LIN {X 0,Y 319.626,Z 323.132,A -85,B 0,C 180,E1 -15102.071,E2 -15102.071} C_VEL
LIN {X 0,Y 319.734,Z 323.151,A -85,B 0,C 180,E1 -15106.008,E2 -15106.008} C_VEL
LIN {X 0,Y 319.737,Z 323.147,A -85,B 0,C 180,E1 -15109.872,E2 -15109.872} C_VEL
LIN {X 0,Y 319.902,Z 323.101,A -85,B 0,C 180,E1 -15113.693,E2 -15113.693} C_VEL
LIN {X 0,Y 319.959,Z 323.12,A -85,B 0,C 180,E1 -15117.482,E2 -15117.482} C_VEL
LIN {X 0,Y 320.015,Z 323.113,A -85,B 0,C 180,E1 -15121.258,E2 -15121.258} C_VEL
LIN {X 0,Y 319.917,Z 323.111,A -85,B 0,C 180,E1 -15126.306,E2 -15126.306} C_VEL
LIN {X 0,Y 319.737,Z 323.154,A -85,B 0,C 180,E1 -15130.127,E2 -15130.127} C_VEL
LIN {X 0,Y 319.71,Z 323.137,A -85,B 0,C 180,E1 -15133.993,E2 -15133.993} C_VEL
LIN {X 0,Y 319.587,Z 323.169,A -85,B 0,C 180,E1 -15137.931,E2 -15137.931} C_VEL
LIN {X 0,Y 319.564,Z 323.172,A -85,B 0,C 180,E1 -15141.954,E2 -15141.954} C_VEL
LIN {X 0,Y 319.567,Z 323.17,A -85,B 0,C 180,E1 -15146.094,E2 -15146.094} C_VEL
LIN {X 0,Y 319.541,Z 323.179,A -85,B 0,C 180,E1 -15148.938,E2 -15148.938} C_VEL
LIN {X 0,Y 319.523,Z 323.172,A -85,B 0,C 180,E1 -15151.862,E2 -15151.862} C_VEL
LIN {X 0,Y 319.579,Z 323.174,A -85,B 0,C 180,E1 -15155.542,E2 -15155.542} C_VEL
LIN {X 0,Y 319.527,Z 323.183,A -85,B 0,C 180,E1 -15159.661,E2 -15159.661} C_VEL
LIN {X 0,Y 319.517,Z 323.178,A -85,B 0,C 180,E1 -15163.459,E2 -15163.459} C_VEL
LIN {X 0,Y 319.548,Z 323.18,A -85,B 0,C 180,E1 -15167.015,E2 -15167.015} C_VEL
LIN {X 0,Y 319.543,Z 323.181,A -85,B 0,C 180,E1 -15170.37,E2 -15170.37} C_VEL
LIN {X 0,Y 319.577,Z 323.176,A -85,B 0,C 180,E1 -15174.457,E2 -15174.457} C_VEL
LIN {X 0,Y 319.522,Z 323.186,A -85,B 0,C 180,E1 -15178.137,E2 -15178.137} C_VEL
LIN {X 0,Y 319.566,Z 323.328,A -85,B 0,C 180,E1 -15179.059,E2 -15179.059} C_VEL
LIN {X 0,Y 321.759,Z 333.663,A -85,B 0,C 180,E1 -15182.344,E2 -15182.344} C_VEL
LIN {X 0,Y 323.542,Z 343.466,A -85,B 0,C 180,E1 -15185.283,E2 -15185.283} C_VEL
LIN {X 0,Y 323.619,Z 344.48,A -85,B 0,C 180,E1 -15185.48,E2 -15185.48} C_VEL
LIN {X 0,Y 328.326,Z 371.476,A -85,B 0,C 180,E1 -15186.494,E2 -15186.494} C_VEL
LIN {X 0,Y 329.76,Z 380.86,A -85,B 0,C 180,E1 -15186.815,E2 -15186.815} C_VEL
LIN {X 0,Y 328.137,Z 450.866,A -85,B 0,C 180,E1 -15188.401,E2 -15188.401} C_VEL
LIN {X 0,Y 327.713,Z 460.449,A -85,B 0,C 180,E1 -15188.742,E2 -15188.742} C_VEL
LIN {X 0,Y 327.027,Z 470.32,A -85,B 0,C 180,E1 -15189.231,E2 -15189.231} C_VEL
LIN {X 0,Y 326.274,Z 479.678,A -85,B 0,C 180,E1 -15189.84,E2 -15189.84} C_VEL
LIN {X 0,Y 325.191,Z 490.522,A -85,B 0,C 180,E1 -15190.756,E2 -15190.756} C_VEL
LIN {X 0,Y 324.039,Z 500.641,A -85,B 0,C 180,E1 -15191.834,E2 -15191.834} C_VEL
LIN {X 0,Y 322.955,Z 509.479,A -85,B 0,C 180,E1 -15192.981,E2 -15192.981} C_VEL
LIN {X 0,Y 321.975,Z 517.57,A -85,B 0,C 180,E1 -15194.242,E2 -15194.242} C_VEL
LIN {X 0,Y 320.934,Z 525.527,A -85,B 0,C 180,E1 -15195.738,E2 -15195.738} C_VEL
LIN {X 0,Y 319.888,Z 532.482,A -85,B 0,C 180,E1 -15197.308,E2 -15197.308} C_VEL
LIN {X 0,Y 319.042,Z 539.265,A -85,B 0,C 180,E1 -15199.208,E2 -15199.208} C_VEL
LIN {X 0,Y 318.623,Z 543.11,A -85,B 0,C 180,E1 -15200.478,E2 -15200.478} C_VEL
LIN {X 0,Y 318.164,Z 547.736,A -85,B 0,C 180,E1 -15202.384,E2 -15202.384} C_VEL
LIN {X 0,Y 317.864,Z 551.156,A -85,B 0,C 180,E1 -15204.237,E2 -15204.237} C_VEL
LIN {X 0,Y 317.772,Z 553.736,A -85,B 0,C 180,E1 -15206.196,E2 -15206.196} C_VEL
LIN {X 0,Y 317.686,Z 555.558,A -85,B 0,C 180,E1 -15208.732,E2 -15208.732} C_VEL
LIN {X 0,Y 317.7,Z 555.874,A -85,B 0,C 180,E1 -15210,E2 -15210} C_VEL
LIN {X 0,Y 317.725,Z 555.365,A -85,B 0,C 180,E1 -15212.535,E2 -15212.535} C_VEL
LIN {X 0,Y 317.843,Z 553.108,A -85,B 0,C 180,E1 -15215.074,E2 -15215.074} C_VEL
LIN {X 0,Y 318.061,Z 550.377,A -85,B 0,C 180,E1 -15216.98,E2 -15216.98} C_VEL
LIN {X 0,Y 318.49,Z 546.623,A -85,B 0,C 180,E1 -15218.886,E2 -15218.886} C_VEL
LIN {X 0,Y 319.153,Z 541.741,A -85,B 0,C 180,E1 -15220.788,E2 -15220.788} C_VEL
LIN {X 0,Y 319.861,Z 536.759,A -85,B 0,C 180,E1 -15222.37,E2 -15222.37} C_VEL
LIN {X 0,Y 321.147,Z 529.338,A -85,B 0,C 180,E1 -15224.252,E2 -15224.252} C_VEL
LIN {X 0,Y 322.305,Z 521.825,A -85,B 0,C 180,E1 -15225.817,E2 -15225.817} C_VEL
LIN {X 0,Y 323.459,Z 513.882,A -85,B 0,C 180,E1 -15227.195,E2 -15227.195} C_VEL
LIN {X 0,Y 324.723,Z 505.12,A -85,B 0,C 180,E1 -15228.453,E2 -15228.453} C_VEL
LIN {X 0,Y 325.995,Z 496.099,A -85,B 0,C 180,E1 -15229.521,E2 -15229.521} C_VEL
LIN {X 0,Y 327.231,Z 486.747,A -85,B 0,C 180,E1 -15230.426,E2 -15230.426} C_VEL
LIN {X 0,Y 328.338,Z 475.986,A -85,B 0,C 180,E1 -15231.256,E2 -15231.256} C_VEL
LIN {X 0,Y 329.341,Z 464.293,A -85,B 0,C 180,E1 -15231.928,E2 -15231.928} C_VEL
LIN {X 0,Y 330.1,Z 453.228,A -85,B 0,C 180,E1 -15232.369,E2 -15232.369} C_VEL
LIN {X 0,Y 330.612,Z 433.555,A -85,B 0,C 180,E1 -15232.868,E2 -15232.868} C_VEL
LIN {X 0,Y 331.874,Z 381.21,A -85,B 0,C 180,E1 -15234.044,E2 -15234.044} C_VEL
LIN {X 0,Y 328.247,Z 359.793,A -85,B 0,C 180,E1 -15234.893,E2 -15234.893} C_VEL
LIN {X 0,Y 325.512,Z 347.56,A -85,B 0,C 180,E1 -15235.451,E2 -15235.451} C_VEL
LIN {X 0,Y 323.992,Z 343.545,A -85,B 0,C 180,E1 -15235.749,E2 -15235.749} C_VEL
LIN {X 0,Y 321.996,Z 333.704,A -85,B 0,C 180,E1 -15238.697,E2 -15238.697} C_VEL
LIN {X 0,Y 319.726,Z 323.984,A -85,B 0,C 180,E1 -15241.84,E2 -15241.84} C_VEL
LIN {X 0,Y 319.563,Z 323.201,A -85,B 0,C 180,E1 -15242.23,E2 -15242.23} C_VEL
LIN {X 0,Y 319.557,Z 323.173,A -85,B 0,C 180,E1 -15246.428,E2 -15246.428} C_VEL
LIN {X 0,Y 319.557,Z 323.169,A -85,B 0,C 180,E1 -15249.669,E2 -15249.669} C_VEL
LIN {X 0,Y 319.519,Z 323.183,A -85,B 0,C 180,E1 -15253.461,E2 -15253.461} C_VEL
LIN {X 0,Y 319.552,Z 323.18,A -85,B 0,C 180,E1 -15257.017,E2 -15257.017} C_VEL
LIN {X 0,Y 319.545,Z 323.179,A -85,B 0,C 180,E1 -15260.371,E2 -15260.371} C_VEL
LIN {X 0,Y 319.578,Z 323.17,A -85,B 0,C 180,E1 -15264.457,E2 -15264.457} C_VEL
LIN {X 0,Y 319.53,Z 323.177,A -85,B 0,C 180,E1 -15268.139,E2 -15268.139} C_VEL
LIN {X 0,Y 319.61,Z 323.169,A -85,B 0,C 180,E1 -15271.591,E2 -15271.591} C_VEL
LIN {X 0,Y 319.605,Z 323.171,A -85,B 0,C 180,E1 -15275.304,E2 -15275.304} C_VEL
LIN {X 0,Y 319.597,Z 323.169,A -85,B 0,C 180,E1 -15278.048,E2 -15278.048} C_VEL
LIN {X 0,Y 319.689,Z 323.156,A -85,B 0,C 180,E1 -15280.962,E2 -15280.962} C_VEL
LIN {X 0,Y 319.731,Z 323.152,A -85,B 0,C 180,E1 -15285.276,E2 -15285.276} C_VEL
LIN {X 0,Y 319.759,Z 323.149,A -85,B 0,C 180,E1 -15289.873,E2 -15289.873} C_VEL
LIN {X 0,Y 319.935,Z 323.13,A -85,B 0,C 180,E1 -15292.427,E2 -15292.427} C_VEL
LIN {X 0,Y 319.749,Z 323.148,A -85,B 0,C 180,E1 -15294.956,E2 -15294.956} C_VEL
LIN {X 0,Y 319.993,Z 323.122,A -85,B 0,C 180,E1 -15297.483,E2 -15297.483} C_VEL
LIN {X 0,Y 320.152,Z 323.098,A -85,B 0,C 180,E1 -15300,E2 -15300} C_VEL
LIN {X 0,Y 319.993,Z 323.125,A -85,B 0,C 180,E1 -15302.518,E2 -15302.518} C_VEL
LIN {X 0,Y 319.934,Z 323.128,A -85,B 0,C 180,E1 -15306.628,E2 -15306.628} C_VEL
LIN {X 0,Y 319.759,Z 323.152,A -85,B 0,C 180,E1 -15310.127,E2 -15310.127} C_VEL
LIN {X 0,Y 319.732,Z 323.156,A -85,B 0,C 180,E1 -15314.724,E2 -15314.724} C_VEL
LIN {X 0,Y 319.69,Z 323.158,A -85,B 0,C 180,E1 -15319.038,E2 -15319.038} C_VEL
LIN {X 0,Y 319.559,Z 323.179,A -85,B 0,C 180,E1 -15323.321,E2 -15323.321} C_VEL
LIN {X 0,Y 319.589,Z 323.175,A -85,B 0,C 180,E1 -15326.092,E2 -15326.092} C_VEL
LIN {X 0,Y 319.576,Z 323.173,A -85,B 0,C 180,E1 -15328.935,E2 -15328.935} C_VEL
LIN {X 0,Y 319.531,Z 323.177,A -85,B 0,C 180,E1 -15331.862,E2 -15331.862} C_VEL
LIN {X 0,Y 319.57,Z 323.179,A -85,B 0,C 180,E1 -15335.54,E2 -15335.54} C_VEL
LIN {X 0,Y 319.649,Z 323.459,A -85,B 0,C 180,E1 -15336.347,E2 -15336.347} C_VEL
LIN {X 0,Y 322.123,Z 333.874,A -85,B 0,C 180,E1 -15339.665,E2 -15339.665} C_VEL
LIN {X 0,Y 322.612,Z 336.041,A -85,B 0,C 180,E1 -15340.207,E2 -15340.207} C_VEL
LIN {X 0,Y 328.68,Z 350.643,A -85,B 0,C 180,E1 -15341.162,E2 -15341.162} C_VEL
LIN {X 0,Y 332.144,Z 368.395,A -85,B 0,C 180,E1 -15341.908,E2 -15341.908} C_VEL
LIN {X 0,Y 330.201,Z 442.436,A -85,B 0,C 180,E1 -15343.6,E2 -15343.6} C_VEL
LIN {X 0,Y 329.689,Z 451.952,A -85,B 0,C 180,E1 -15343.936,E2 -15343.936} C_VEL
LIN {X 0,Y 329.089,Z 461.748,A -85,B 0,C 180,E1 -15344.432,E2 -15344.432} C_VEL
LIN {X 0,Y 328.119,Z 472.227,A -85,B 0,C 180,E1 -15345.131,E2 -15345.131} C_VEL
LIN {X 0,Y 327.138,Z 481.657,A -85,B 0,C 180,E1 -15345.931,E2 -15345.931} C_VEL
LIN {X 0,Y 325.754,Z 492.603,A -85,B 0,C 180,E1 -15347.108,E2 -15347.108} C_VEL
LIN {X 0,Y 324.528,Z 501.273,A -85,B 0,C 180,E1 -15348.247,E2 -15348.247} C_VEL
LIN {X 0,Y 323.167,Z 509.632,A -85,B 0,C 180,E1 -15349.566,E2 -15349.566} C_VEL
LIN {X 0,Y 321.945,Z 517.518,A -85,B 0,C 180,E1 -15351.082,E2 -15351.082} C_VEL
LIN {X 0,Y 320.914,Z 524.004,A -85,B 0,C 180,E1 -15352.575,E2 -15352.575} C_VEL
LIN {X 0,Y 319.836,Z 530.455,A -85,B 0,C 180,E1 -15354.393,E2 -15354.393} C_VEL
LIN {X 0,Y 319.231,Z 534.761,A -85,B 0,C 180,E1 -15355.848,E2 -15355.848} C_VEL
LIN {X 0,Y 318.47,Z 539.726,A -85,B 0,C 180,E1 -15358.02,E2 -15358.02} C_VEL
LIN {X 0,Y 318.152,Z 542.372,A -85,B 0,C 180,E1 -15359.487,E2 -15359.487} C_VEL
LIN {X 0,Y 317.871,Z 544.215,A -85,B 0,C 180,E1 -15360.895,E2 -15360.895} C_VEL
LIN {X 0,Y 317.665,Z 545.633,A -85,B 0,C 180,E1 -15362.316,E2 -15362.316} C_VEL
LIN {X 0,Y 317.493,Z 546.626,A -85,B 0,C 180,E1 -15363.723,E2 -15363.723} C_VEL
LIN {X 0,Y 317.423,Z 546.993,A -85,B 0,C 180,E1 -15365.2,E2 -15365.2} C_VEL
LIN {X 0,Y 317.434,Z 546.413,A -85,B 0,C 180,E1 -15367.89,E2 -15367.89} C_VEL
LIN {X 0,Y 317.593,Z 545.359,A -85,B 0,C 180,E1 -15369.264,E2 -15369.264} C_VEL
LIN {X 0,Y 317.987,Z 541.947,A -85,B 0,C 180,E1 -15371.976,E2 -15371.976} C_VEL
LIN {X 0,Y 318.387,Z 538.074,A -85,B 0,C 180,E1 -15373.983,E2 -15373.983} C_VEL
LIN {X 0,Y 318.979,Z 532.982,A -85,B 0,C 180,E1 -15375.974,E2 -15375.974} C_VEL
LIN {X 0,Y 319.643,Z 527.744,A -85,B 0,C 180,E1 -15377.621,E2 -15377.621} C_VEL
LIN {X 0,Y 320.481,Z 521.404,A -85,B 0,C 180,E1 -15379.257,E2 -15379.257} C_VEL
LIN {X 0,Y 321.607,Z 513.482,A -85,B 0,C 180,E1 -15380.922,E2 -15380.922} C_VEL
LIN {X 0,Y 322.656,Z 505.376,A -85,B 0,C 180,E1 -15382.333,E2 -15382.333} C_VEL
LIN {X 0,Y 323.8,Z 496.471,A -85,B 0,C 180,E1 -15383.614,E2 -15383.614} C_VEL
LIN {X 0,Y 324.744,Z 488.557,A -85,B 0,C 180,E1 -15384.573,E2 -15384.573} C_VEL
LIN {X 0,Y 325.898,Z 477.255,A -85,B 0,C 180,E1 -15385.671,E2 -15385.671} C_VEL
LIN {X 0,Y 326.86,Z 466.957,A -85,B 0,C 180,E1 -15386.456,E2 -15386.456} C_VEL
LIN {X 0,Y 327.52,Z 456.409,A -85,B 0,C 180,E1 -15387.079,E2 -15387.079} C_VEL
LIN {X 0,Y 328.185,Z 445.003,A -85,B 0,C 180,E1 -15387.545,E2 -15387.545} C_VEL
LIN {X 0,Y 328.673,Z 428.296,A -85,B 0,C 180,E1 -15387.971,E2 -15387.971} C_VEL
LIN {X 0,Y 329.901,Z 367.398,A -85,B 0,C 180,E1 -15389.329,E2 -15389.329} C_VEL
LIN {X 0,Y 325.686,Z 345.307,A -85,B 0,C 180,E1 -15390.151,E2 -15390.151} C_VEL
LIN {X 0,Y 322.567,Z 336.108,A -85,B 0,C 180,E1 -15390.648,E2 -15390.648} C_VEL
LIN {X 0,Y 320.926,Z 328.238,A -85,B 0,C 180,E1 -15393.139,E2 -15393.139} C_VEL
LIN {X 0,Y 319.738,Z 323.207,A -85,B 0,C 180,E1 -15394.886,E2 -15394.886} C_VEL
LIN {X 0,Y 319.937,Z 323.128,A -85,B 0,C 180,E1 -15396.306,E2 -15396.306} C_VEL
LIN {X 0,Y 319.737,Z 323.157,A -85,B 0,C 180,E1 -15400.128,E2 -15400.128} C_VEL
LIN {X 0,Y 319.734,Z 323.158,A -85,B 0,C 180,E1 -15403.992,E2 -15403.992} C_VEL
LIN {X 0,Y 319.66,Z 323.165,A -85,B 0,C 180,E1 -15407.927,E2 -15407.927} C_VEL
LIN {X 0,Y 319.605,Z 323.176,A -85,B 0,C 180,E1 -15410.6,E2 -15410.6} C_VEL
LIN {X 0,Y 319.606,Z 323.171,A -85,B 0,C 180,E1 -15414.696,E2 -15414.696} C_VEL
LIN {X 0,Y 319.613,Z 323.16,A -85,B 0,C 180,E1 -15418.41,E2 -15418.41} C_VEL
LIN {X 0,Y 319.532,Z 323.179,A -85,B 0,C 180,E1 -15421.862,E2 -15421.862} C_VEL
LIN {X 0,Y 319.548,Z 323.162,A -85,B 0,C 180,E1 -15424.612,E2 -15424.612} C_VEL
LIN {X 0,Y 318.92,Z 323.25,A -85,B 0,C 180,E1 -15425.664,E2 -15425.664} C_VEL
LIN {X 0,Y 316.093,Z 323.61,A -85,B 0,C 180,E1 -15427.378,E2 -15427.378} C_VEL
LIN {X 0,Y 313.662,Z 323.912,A -85,B 0,C 180,E1 -15428.766,E2 -15428.766} C_VEL
LIN {X 0,Y 312.598,Z 324.039,A -85,B 0,C 180,E1 -15429.841,E2 -15429.841} C_VEL
LIN {X 0,Y 312.502,Z 324.045,A -85,B 0,C 180,E1 -15430.206,E2 -15430.206} C_VEL
LIN {X 0,Y 312.475,Z 324.055,A -85,B 0,C 180,E1 -15434.206,E2 -15434.206} C_VEL
LIN {X 0,Y 312.486,Z 324.053,A -85,B 0,C 180,E1 -15437.919,E2 -15437.919} C_VEL
LIN {X 0,Y 312.479,Z 324.035,A -85,B 0,C 180,E1 -15440.968,E2 -15440.968} C_VEL
LIN {X 0,Y 312.533,Z 324.05,A -85,B 0,C 180,E1 -15444.22,E2 -15444.22} C_VEL
LIN {X 0,Y 312.503,Z 324.052,A -85,B 0,C 180,E1 -15447.333,E2 -15447.333} C_VEL
LIN {X 0,Y 312.509,Z 324.024,A -85,B 0,C 180,E1 -15451.291,E2 -15451.291} C_VEL
LIN {X 0,Y 312.556,Z 324.049,A -85,B 0,C 180,E1 -15454.708,E2 -15454.708} C_VEL
LIN {X 0,Y 312.568,Z 324.045,A -85,B 0,C 180,E1 -15457.527,E2 -15457.527} C_VEL
LIN {X 0,Y 312.584,Z 324.008,A -85,B 0,C 180,E1 -15461.653,E2 -15461.653} C_VEL
LIN {X 0,Y 312.688,Z 324.03,A -85,B 0,C 180,E1 -15465.686,E2 -15465.686} C_VEL
LIN {X 0,Y 312.687,Z 324.028,A -85,B 0,C 180,E1 -15469.641,E2 -15469.641} C_VEL
LIN {X 0,Y 312.798,Z 323.991,A -85,B 0,C 180,E1 -15472.252,E2 -15472.252} C_VEL
LIN {X 0,Y 312.692,Z 324.007,A -85,B 0,C 180,E1 -15474.842,E2 -15474.842} C_VEL
LIN {X 0,Y 312.969,Z 323.998,A -85,B 0,C 180,E1 -15478.713,E2 -15478.713} C_VEL
LIN {X 0,Y 312.982,Z 323.989,A -85,B 0,C 180,E1 -15481.286,E2 -15481.286} C_VEL
LIN {X 0,Y 312.86,Z 323.99,A -85,B 0,C 180,E1 -15486.449,E2 -15486.449} C_VEL
LIN {X 0,Y 312.752,Z 324.024,A -85,B 0,C 180,E1 -15489.05,E2 -15489.05} C_VEL
LIN {X 0,Y 312.626,Z 324.033,A -85,B 0,C 180,E1 -15492.991,E2 -15492.991} C_VEL
LIN {X 0,Y 312.57,Z 324.024,A -85,B 0,C 180,E1 -15495.653,E2 -15495.653} C_VEL
LIN {X 0,Y 312.534,Z 324.054,A -85,B 0,C 180,E1 -15499.712,E2 -15499.712} C_VEL
LIN {X 0,Y 312.521,Z 324.038,A -85,B 0,C 180,E1 -15502.777,E2 -15502.777} C_VEL
LIN {X 0,Y 312.528,Z 324.046,A -85,B 0,C 180,E1 -15505.907,E2 -15505.907} C_VEL
LIN {X 0,Y 312.495,Z 324.05,A -85,B 0,C 180,E1 -15509.655,E2 -15509.655} C_VEL
LIN {X 0,Y 312.519,Z 324.058,A -85,B 0,C 180,E1 -15513.688,E2 -15513.688} C_VEL
LIN {X 0,Y 312.51,Z 324.046,A -85,B 0,C 180,E1 -15517.387,E2 -15517.387} C_VEL
LIN {X 0,Y 312.439,Z 324.063,A -85,B 0,C 180,E1 -15520.717,E2 -15520.717} C_VEL
LIN {X 0,Y 312.448,Z 324.065,A -85,B 0,C 180,E1 -15524.21,E2 -15524.21} C_VEL
LIN {X 0,Y 312.452,Z 324.064,A -85,B 0,C 180,E1 -15527.925,E2 -15527.925} C_VEL
LIN {X 0,Y 312.482,Z 324.058,A -85,B 0,C 180,E1 -15531.922,E2 -15531.922} C_VEL
LIN {X 0,Y 312.528,Z 324.054,A -85,B 0,C 180,E1 -15534.22,E2 -15534.22} C_VEL
LIN {X 0,Y 312.476,Z 324.064,A -85,B 0,C 180,E1 -15538.088,E2 -15538.088} C_VEL
LIN {X 0,Y 312.525,Z 324.325,A -85,B 0,C 180,E1 -15538.708,E2 -15538.708} C_VEL
LIN {X 0,Y 314.721,Z 334.563,A -85,B 0,C 180,E1 -15542.034,E2 -15542.034} C_VEL
LIN {X 0,Y 316.54,Z 344.066,A -85,B 0,C 180,E1 -15544.917,E2 -15544.917} C_VEL
LIN {X 0,Y 317.353,Z 347.388,A -85,B 0,C 180,E1 -15545.128,E2 -15545.128} C_VEL
LIN {X 0,Y 322.634,Z 377.952,A -85,B 0,C 180,E1 -15546.256,E2 -15546.256} C_VEL
LIN {X 0,Y 323.125,Z 381.869,A -85,B 0,C 180,E1 -15546.386,E2 -15546.386} C_VEL
LIN {X 0,Y 321.461,Z 450.859,A -85,B 0,C 180,E1 -15547.982,E2 -15547.982} C_VEL
LIN {X 0,Y 321.033,Z 460.207,A -85,B 0,C 180,E1 -15548.32,E2 -15548.32} C_VEL
LIN {X 0,Y 320.267,Z 470.718,A -85,B 0,C 180,E1 -15548.856,E2 -15548.856} C_VEL
LIN {X 0,Y 319.396,Z 480.902,A -85,B 0,C 180,E1 -15549.554,E2 -15549.554} C_VEL
LIN {X 0,Y 318.295,Z 491.487,A -85,B 0,C 180,E1 -15550.49,E2 -15550.49} C_VEL
LIN {X 0,Y 317.092,Z 501.414,A -85,B 0,C 180,E1 -15551.589,E2 -15551.589} C_VEL
LIN {X 0,Y 316.054,Z 509.696,A -85,B 0,C 180,E1 -15552.697,E2 -15552.697} C_VEL
LIN {X 0,Y 315.051,Z 517.587,A -85,B 0,C 180,E1 -15553.958,E2 -15553.958} C_VEL
LIN {X 0,Y 314.017,Z 525.219,A -85,B 0,C 180,E1 -15555.417,E2 -15555.417} C_VEL
LIN {X 0,Y 312.953,Z 532.212,A -85,B 0,C 180,E1 -15557.022,E2 -15557.022} C_VEL
LIN {X 0,Y 312.047,Z 539.027,A -85,B 0,C 180,E1 -15558.963,E2 -15558.963} C_VEL
LIN {X 0,Y 311.408,Z 544.485,A -85,B 0,C 180,E1 -15560.91,E2 -15560.91} C_VEL
LIN {X 0,Y 310.95,Z 548.753,A -85,B 0,C 180,E1 -15562.859,E2 -15562.859} C_VEL
LIN {X 0,Y 310.719,Z 551.951,A -85,B 0,C 180,E1 -15564.809,E2 -15564.809} C_VEL
LIN {X 0,Y 310.687,Z 553.581,A -85,B 0,C 180,E1 -15566.109,E2 -15566.109} C_VEL
LIN {X 0,Y 310.603,Z 555.448,A -85,B 0,C 180,E1 -15568.703,E2 -15568.703} C_VEL
LIN {X 0,Y 310.614,Z 555.764,A -85,B 0,C 180,E1 -15570,E2 -15570} C_VEL
LIN {X 0,Y 310.651,Z 555.291,A -85,B 0,C 180,E1 -15572.593,E2 -15572.593} C_VEL
LIN {X 0,Y 310.763,Z 553.062,A -85,B 0,C 180,E1 -15575.19,E2 -15575.19} C_VEL
LIN {X 0,Y 311.003,Z 550.354,A -85,B 0,C 180,E1 -15577.14,E2 -15577.14} C_VEL
LIN {X 0,Y 311.449,Z 546.623,A -85,B 0,C 180,E1 -15579.088,E2 -15579.088} C_VEL
LIN {X 0,Y 312.165,Z 541.766,A -85,B 0,C 180,E1 -15581.032,E2 -15581.032} C_VEL
LIN {X 0,Y 312.908,Z 536.811,A -85,B 0,C 180,E1 -15582.649,E2 -15582.649} C_VEL
LIN {X 0,Y 314.25,Z 529.419,A -85,B 0,C 180,E1 -15584.572,E2 -15584.572} C_VEL
LIN {X 0,Y 315.459,Z 521.95,A -85,B 0,C 180,E1 -15586.17,E2 -15586.17} C_VEL
LIN {X 0,Y 316.716,Z 513.909,A -85,B 0,C 180,E1 -15587.598,E2 -15587.598} C_VEL
LIN {X 0,Y 318.014,Z 505.371,A -85,B 0,C 180,E1 -15588.857,E2 -15588.857} C_VEL
LIN {X 0,Y 319.334,Z 496.44,A -85,B 0,C 180,E1 -15589.946,E2 -15589.946} C_VEL
LIN {X 0,Y 320.623,Z 487.211,A -85,B 0,C 180,E1 -15590.867,E2 -15590.867} C_VEL
LIN {X 0,Y 321.857,Z 475.424,A -85,B 0,C 180,E1 -15591.79,E2 -15591.79} C_VEL
LIN {X 0,Y 322.852,Z 464.382,A -85,B 0,C 180,E1 -15592.435,E2 -15592.435} C_VEL
LIN {X 0,Y 323.661,Z 453.42,A -85,B 0,C 180,E1 -15592.881,E2 -15592.881} C_VEL
LIN {X 0,Y 324.195,Z 434.067,A -85,B 0,C 180,E1 -15593.385,E2 -15593.385} C_VEL
LIN {X 0,Y 325.509,Z 382.081,A -85,B 0,C 180,E1 -15594.575,E2 -15594.575} C_VEL
LIN {X 0,Y 321.867,Z 360.709,A -85,B 0,C 180,E1 -15595.451,E2 -15595.451} C_VEL
LIN {X 0,Y 319.441,Z 350.024,A -85,B 0,C 180,E1 -15595.96,E2 -15595.96} C_VEL
LIN {X 0,Y 316.817,Z 343.596,A -85,B 0,C 180,E1 -15596.426,E2 -15596.426} C_VEL
LIN {X 0,Y 315.612,Z 337.505,A -85,B 0,C 180,E1 -15598.242,E2 -15598.242} C_VEL
LIN {X 0,Y 313.325,Z 327.475,A -85,B 0,C 180,E1 -15601.532,E2 -15601.532} C_VEL
LIN {X 0,Y 312.542,Z 324.09,A -85,B 0,C 180,E1 -15602.79,E2 -15602.79} C_VEL
LIN {X 0,Y 312.534,Z 324.051,A -85,B 0,C 180,E1 -15605.95,E2 -15605.95} C_VEL
LIN {X 0,Y 312.502,Z 324.046,A -85,B 0,C 180,E1 -15610.126,E2 -15610.126} C_VEL
LIN {X 0,Y 312.456,Z 324.064,A -85,B 0,C 180,E1 -15613.965,E2 -15613.965} C_VEL
LIN {X 0,Y 312.482,Z 324.056,A -85,B 0,C 180,E1 -15617.919,E2 -15617.919} C_VEL
LIN {X 0,Y 312.497,Z 324.056,A -85,B 0,C 180,E1 -15620.971,E2 -15620.971} C_VEL
LIN {X 0,Y 312.531,Z 324.049,A -85,B 0,C 180,E1 -15624.221,E2 -15624.221} C_VEL
LIN {X 0,Y 312.503,Z 324.057,A -85,B 0,C 180,E1 -15627.334,E2 -15627.334} C_VEL
LIN {X 0,Y 312.543,Z 324.05,A -85,B 0,C 180,E1 -15631.279,E2 -15631.279} C_VEL
LIN {X 0,Y 312.585,Z 324.05,A -85,B 0,C 180,E1 -15634.711,E2 -15634.711} C_VEL
LIN {X 0,Y 312.587,Z 324.041,A -85,B 0,C 180,E1 -15637.529,E2 -15637.529} C_VEL
LIN {X 0,Y 312.639,Z 324.031,A -85,B 0,C 180,E1 -15641.657,E2 -15641.657} C_VEL
LIN {X 0,Y 312.694,Z 324.024,A -85,B 0,C 180,E1 -15645.687,E2 -15645.687} C_VEL
LIN {X 0,Y 312.703,Z 324.03,A -85,B 0,C 180,E1 -15649.642,E2 -15649.642} C_VEL
LIN {X 0,Y 312.875,Z 324.007,A -85,B 0,C 180,E1 -15652.255,E2 -15652.255} C_VEL
LIN {X 0,Y 312.719,Z 324.024,A -85,B 0,C 180,E1 -15654.843,E2 -15654.843} C_VEL
LIN {X 0,Y 312.992,Z 323.995,A -85,B 0,C 180,E1 -15658.714,E2 -15658.714} C_VEL
LIN {X 0,Y 312.992,Z 323.992,A -85,B 0,C 180,E1 -15661.287,E2 -15661.287} C_VEL
LIN {X 0,Y 312.719,Z 324.024,A -85,B 0,C 180,E1 -15665.158,E2 -15665.158} C_VEL
LIN {X 0,Y 312.874,Z 324.008,A -85,B 0,C 180,E1 -15667.746,E2 -15667.746} C_VEL
LIN {X 0,Y 312.671,Z 324.033,A -85,B 0,C 180,E1 -15671.672,E2 -15671.672} C_VEL
LIN {X 0,Y 312.701,Z 324.033,A -85,B 0,C 180,E1 -15674.888,E2 -15674.888} C_VEL
LIN {X 0,Y 312.61,Z 324.039,A -85,B 0,C 180,E1 -15679.225,E2 -15679.225} C_VEL
LIN {X 0,Y 312.526,Z 324.056,A -85,B 0,C 180,E1 -15682.78,E2 -15682.78} C_VEL
LIN {X 0,Y 312.569,Z 324.052,A -85,B 0,C 180,E1 -15685.923,E2 -15685.923} C_VEL
LIN {X 0,Y 312.537,Z 324.055,A -85,B 0,C 180,E1 -15689.651,E2 -15689.651} C_VEL
LIN {X 0,Y 312.52,Z 324.051,A -85,B 0,C 180,E1 -15693.689,E2 -15693.689} C_VEL
LIN {X 0,Y 312.565,Z 324.201,A -85,B 0,C 180,E1 -15695.676,E2 -15695.676} C_VEL
LIN {X 0,Y 315.023,Z 334.395,A -85,B 0,C 180,E1 -15699.068,E2 -15699.068} C_VEL
LIN {X 0,Y 315.399,Z 335.975,A -85,B 0,C 180,E1 -15699.477,E2 -15699.477} C_VEL
LIN {X 0,Y 322.335,Z 352.441,A -85,B 0,C 180,E1 -15700.625,E2 -15700.625} C_VEL
LIN {X 0,Y 325.131,Z 365.615,A -85,B 0,C 180,E1 -15701.22,E2 -15701.22} C_VEL
LIN {X 0,Y 325.83,Z 369.74,A -85,B 0,C 180,E1 -15701.387,E2 -15701.387} C_VEL
LIN {X 0,Y 323.775,Z 442.238,A -85,B 0,C 180,E1 -15703.067,E2 -15703.067} C_VEL
LIN {X 0,Y 323.231,Z 452.055,A -85,B 0,C 180,E1 -15703.419,E2 -15703.419} C_VEL
LIN {X 0,Y 322.593,Z 461.823,A -85,B 0,C 180,E1 -15703.921,E2 -15703.921} C_VEL
LIN {X 0,Y 321.701,Z 471.566,A -85,B 0,C 180,E1 -15704.573,E2 -15704.573} C_VEL
LIN {X 0,Y 320.586,Z 481.765,A -85,B 0,C 180,E1 -15705.451,E2 -15705.451} C_VEL
LIN {X 0,Y 319.172,Z 492.366,A -85,B 0,C 180,E1 -15706.606,E2 -15706.606} C_VEL
LIN {X 0,Y 317.843,Z 501.346,A -85,B 0,C 180,E1 -15707.807,E2 -15707.807} C_VEL
LIN {X 0,Y 316.311,Z 510.289,A -85,B 0,C 180,E1 -15709.261,E2 -15709.261} C_VEL
LIN {X 0,Y 315.25,Z 516.942,A -85,B 0,C 180,E1 -15710.553,E2 -15710.553} C_VEL
LIN {X 0,Y 313.922,Z 524.741,A -85,B 0,C 180,E1 -15712.406,E2 -15712.406} C_VEL
LIN {X 0,Y 312.826,Z 531.059,A -85,B 0,C 180,E1 -15714.259,E2 -15714.259} C_VEL
LIN {X 0,Y 312.174,Z 535.277,A -85,B 0,C 180,E1 -15715.749,E2 -15715.749} C_VEL
LIN {X 0,Y 311.636,Z 538.738,A -85,B 0,C 180,E1 -15717.232,E2 -15717.232} C_VEL
LIN {X 0,Y 311.126,Z 542.2,A -85,B 0,C 180,E1 -15719.135,E2 -15719.135} C_VEL
LIN {X 0,Y 310.623,Z 545.547,A -85,B 0,C 180,E1 -15721.933,E2 -15721.933} C_VEL
LIN {X 0,Y 310.452,Z 546.391,A -85,B 0,C 180,E1 -15723.079,E2 -15723.079} C_VEL
LIN {X 0,Y 310.35,Z 547.044,A -85,B 0,C 180,E1 -15724.934,E2 -15724.934} C_VEL
LIN {X 0,Y 310.3,Z 546.754,A -85,B 0,C 180,E1 -15727.354,E2 -15727.354} C_VEL
LIN {X 0,Y 310.599,Z 544.597,A -85,B 0,C 180,E1 -15730.159,E2 -15730.159} C_VEL
LIN {X 0,Y 310.951,Z 541.588,A -85,B 0,C 180,E1 -15732.322,E2 -15732.322} C_VEL
LIN {X 0,Y 311.374,Z 537.779,A -85,B 0,C 180,E1 -15734.285,E2 -15734.285} C_VEL
LIN {X 0,Y 311.802,Z 534.276,A -85,B 0,C 180,E1 -15735.747,E2 -15735.747} C_VEL
LIN {X 0,Y 312.566,Z 528.465,A -85,B 0,C 180,E1 -15737.666,E2 -15737.666} C_VEL
LIN {X 0,Y 313.63,Z 520.77,A -85,B 0,C 180,E1 -15739.673,E2 -15739.673} C_VEL
LIN {X 0,Y 314.517,Z 514.697,A -85,B 0,C 180,E1 -15741.001,E2 -15741.001} C_VEL
LIN {X 0,Y 315.774,Z 505.488,A -85,B 0,C 180,E1 -15742.648,E2 -15742.648} C_VEL
LIN {X 0,Y 316.956,Z 496.761,A -85,B 0,C 180,E1 -15743.931,E2 -15743.931} C_VEL
LIN {X 0,Y 318.078,Z 487.201,A -85,B 0,C 180,E1 -15745.089,E2 -15745.089} C_VEL
LIN {X 0,Y 319.128,Z 477.377,A -85,B 0,C 180,E1 -15746.054,E2 -15746.054} C_VEL
LIN {X 0,Y 320.132,Z 467.076,A -85,B 0,C 180,E1 -15746.854,E2 -15746.854} C_VEL
LIN {X 0,Y 320.831,Z 456.518,A -85,B 0,C 180,E1 -15747.489,E2 -15747.489} C_VEL
LIN {X 0,Y 321.505,Z 445.146,A -85,B 0,C 180,E1 -15747.964,E2 -15747.964} C_VEL
LIN {X 0,Y 322.033,Z 426.774,A -85,B 0,C 180,E1 -15748.437,E2 -15748.437} C_VEL
LIN {X 0,Y 323.291,Z 368.33,A -85,B 0,C 180,E1 -15749.766,E2 -15749.766} C_VEL
LIN {X 0,Y 319.248,Z 347.258,A -85,B 0,C 180,E1 -15750.578,E2 -15750.578} C_VEL
LIN {X 0,Y 315.355,Z 336.451,A -85,B 0,C 180,E1 -15751.178,E2 -15751.178} C_VEL
LIN {X 0,Y 314.869,Z 333.805,A -85,B 0,C 180,E1 -15751.919,E2 -15751.919} C_VEL
LIN {X 0,Y 312.739,Z 324.079,A -85,B 0,C 180,E1 -15755.279,E2 -15755.279} C_VEL
LIN {X 0,Y 312.832,Z 324.013,A -85,B 0,C 180,E1 -15757.747,E2 -15757.747} C_VEL
LIN {X 0,Y 312.665,Z 324.029,A -85,B 0,C 180,E1 -15761.672,E2 -15761.672} C_VEL
LIN {X 0,Y 312.702,Z 324.03,A -85,B 0,C 180,E1 -15764.888,E2 -15764.888} C_VEL
LIN {X 0,Y 312.611,Z 324.036,A -85,B 0,C 180,E1 -15769.225,E2 -15769.225} C_VEL
LIN {X 0,Y 312.53,Z 324.046,A -85,B 0,C 180,E1 -15772.781,E2 -15772.781} C_VEL
LIN {X 0,Y 312.604,Z 324.044,A -85,B 0,C 180,E1 -15775.935,E2 -15775.935} C_VEL
LIN {X 0,Y 312.54,Z 324.051,A -85,B 0,C 180,E1 -15779.651,E2 -15779.651} C_VEL
LIN {X 0,Y 312.521,Z 324.04,A -85,B 0,C 180,E1 -15783.689,E2 -15783.689} C_VEL
LIN {X 0,Y 312.539,Z 324.053,A -85,B 0,C 180,E1 -15787.384,E2 -15787.384} C_VEL
LIN {X 0,Y 312.502,Z 324.045,A -85,B 0,C 180,E1 -15790.206,E2 -15790.206} C_VEL
LIN {X 0,Y 311.802,Z 324.127,A -85,B 0,C 180,E1 -15791.282,E2 -15791.282} C_VEL
LIN {X 0,Y 308.92,Z 324.493,A -85,B 0,C 180,E1 -15793.033,E2 -15793.033} C_VEL
LIN {X 0,Y 306.508,Z 324.801,A -85,B 0,C 180,E1 -15794.453,E2 -15794.453} C_VEL
LIN {X 0,Y 305.495,Z 324.929,A -85,B 0,C 180,E1 -15795.553,E2 -15795.553} C_VEL
LIN {X 0,Y 305.424,Z 324.938,A -85,B 0,C 180,E1 -15795.925,E2 -15795.925} C_VEL
LIN {X 0,Y 305.458,Z 324.91,A -85,B 0,C 180,E1 -15799.892,E2 -15799.892} C_VEL
LIN {X 0,Y 305.481,Z 324.93,A -85,B 0,C 180,E1 -15803.632,E2 -15803.632} C_VEL
LIN {X 0,Y 305.467,Z 324.93,A -85,B 0,C 180,E1 -15806.483,E2 -15806.483} C_VEL
LIN {X 0,Y 305.432,Z 324.909,A -85,B 0,C 180,E1 -15809.587,E2 -15809.587} C_VEL
LIN {X 0,Y 305.462,Z 324.918,A -85,B 0,C 180,E1 -15812.603,E2 -15812.603} C_VEL
LIN {X 0,Y 305.491,Z 324.928,A -85,B 0,C 180,E1 -15815.537,E2 -15815.537} C_VEL
LIN {X 0,Y 305.498,Z 324.913,A -85,B 0,C 180,E1 -15819.813,E2 -15819.813} C_VEL
LIN {X 0,Y 305.546,Z 324.886,A -85,B 0,C 180,E1 -15822.601,E2 -15822.601} C_VEL
LIN {X 0,Y 305.629,Z 324.905,A -85,B 0,C 180,E1 -15825.348,E2 -15825.348} C_VEL
LIN {X 0,Y 305.626,Z 324.91,A -85,B 0,C 180,E1 -15829.399,E2 -15829.399} C_VEL
LIN {X 0,Y 305.748,Z 324.87,A -85,B 0,C 180,E1 -15832.072,E2 -15832.072} C_VEL
LIN {X 0,Y 305.661,Z 324.88,A -85,B 0,C 180,E1 -15834.723,E2 -15834.723} C_VEL
LIN {X 0,Y 305.938,Z 324.874,A -85,B 0,C 180,E1 -15838.683,E2 -15838.683} C_VEL
LIN {X 0,Y 305.948,Z 324.865,A -85,B 0,C 180,E1 -15841.316,E2 -15841.316} C_VEL
LIN {X 0,Y 305.806,Z 324.87,A -85,B 0,C 180,E1 -15846.598,E2 -15846.598} C_VEL
LIN {X 0,Y 305.696,Z 324.906,A -85,B 0,C 180,E1 -15849.261,E2 -15849.261} C_VEL
LIN {X 0,Y 305.573,Z 324.905,A -85,B 0,C 180,E1 -15853.296,E2 -15853.296} C_VEL
LIN {X 0,Y 305.514,Z 324.905,A -85,B 0,C 180,E1 -15856.024,E2 -15856.024} C_VEL
LIN {X 0,Y 305.48,Z 324.934,A -85,B 0,C 180,E1 -15860.187,E2 -15860.187} C_VEL
LIN {X 0,Y 305.487,Z 324.912,A -85,B 0,C 180,E1 -15863.039,E2 -15863.039} C_VEL
LIN {X 0,Y 305.467,Z 324.927,A -85,B 0,C 180,E1 -15866.196,E2 -15866.196} C_VEL
LIN {X 0,Y 305.447,Z 324.933,A -85,B 0,C 180,E1 -15869.033,E2 -15869.033} C_VEL
LIN {X 0,Y 305.436,Z 324.926,A -85,B 0,C 180,E1 -15871.953,E2 -15871.953} C_VEL
LIN {X 0,Y 305.461,Z 324.937,A -85,B 0,C 180,E1 -15875.113,E2 -15875.113} C_VEL
LIN {X 0,Y 305.41,Z 324.937,A -85,B 0,C 180,E1 -15878.519,E2 -15878.519} C_VEL
LIN {X 0,Y 305.432,Z 324.93,A -85,B 0,C 180,E1 -15882.581,E2 -15882.581} C_VEL
LIN {X 0,Y 305.419,Z 324.937,A -85,B 0,C 180,E1 -15886.343,E2 -15886.343} C_VEL
LIN {X 0,Y 305.408,Z 324.94,A -85,B 0,C 180,E1 -15889.884,E2 -15889.884} C_VEL
LIN {X 0,Y 305.461,Z 324.934,A -85,B 0,C 180,E1 -15893.636,E2 -15893.636} C_VEL
LIN {X 0,Y 305.463,Z 324.926,A -85,B 0,C 180,E1 -15896.483,E2 -15896.483} C_VEL
LIN {X 0,Y 305.471,Z 325.175,A -85,B 0,C 180,E1 -15898.267,E2 -15898.267} C_VEL
LIN {X 0,Y 307.419,Z 334.238,A -85,B 0,C 180,E1 -15901.309,E2 -15901.309} C_VEL
LIN {X 0,Y 309.374,Z 344.058,A -85,B 0,C 180,E1 -15904.367,E2 -15904.367} C_VEL
LIN {X 0,Y 310.849,Z 348.756,A -85,B 0,C 180,E1 -15904.665,E2 -15904.665} C_VEL
LIN {X 0,Y 316.19,Z 379.891,A -85,B 0,C 180,E1 -15905.844,E2 -15905.844} C_VEL
LIN {X 0,Y 316.464,Z 385.33,A -85,B 0,C 180,E1 -15905.998,E2 -15905.998} C_VEL
LIN {X 0,Y 314.809,Z 450.747,A -85,B 0,C 180,E1 -15907.542,E2 -15907.542} C_VEL
LIN {X 0,Y 314.366,Z 459.962,A -85,B 0,C 180,E1 -15907.879,E2 -15907.879} C_VEL
LIN {X 0,Y 313.624,Z 469.907,A -85,B 0,C 180,E1 -15908.386,E2 -15908.386} C_VEL
LIN {X 0,Y 312.704,Z 480.248,A -85,B 0,C 180,E1 -15909.097,E2 -15909.097} C_VEL
LIN {X 0,Y 311.589,Z 490.945,A -85,B 0,C 180,E1 -15910.053,E2 -15910.053} C_VEL
LIN {X 0,Y 310.336,Z 500.951,A -85,B 0,C 180,E1 -15911.173,E2 -15911.173} C_VEL
LIN {X 0,Y 309.098,Z 510.323,A -85,B 0,C 180,E1 -15912.466,E2 -15912.466} C_VEL
LIN {X 0,Y 307.983,Z 518.725,A -85,B 0,C 180,E1 -15913.875,E2 -15913.875} C_VEL
LIN {X 0,Y 306.873,Z 526.341,A -85,B 0,C 180,E1 -15915.409,E2 -15915.409} C_VEL
LIN {X 0,Y 305.79,Z 533.123,A -85,B 0,C 180,E1 -15917.051,E2 -15917.051} C_VEL
LIN {X 0,Y 305.062,Z 538.789,A -85,B 0,C 180,E1 -15918.707,E2 -15918.707} C_VEL
LIN {X 0,Y 304.357,Z 544.275,A -85,B 0,C 180,E1 -15920.698,E2 -15920.698} C_VEL
LIN {X 0,Y 303.905,Z 548.571,A -85,B 0,C 180,E1 -15922.693,E2 -15922.693} C_VEL
LIN {X 0,Y 303.634,Z 551.794,A -85,B 0,C 180,E1 -15924.688,E2 -15924.688} C_VEL
LIN {X 0,Y 303.585,Z 553.424,A -85,B 0,C 180,E1 -15926.017,E2 -15926.017} C_VEL
LIN {X 0,Y 303.523,Z 555.337,A -85,B 0,C 180,E1 -15928.673,E2 -15928.673} C_VEL
LIN {X 0,Y 303.53,Z 555.653,A -85,B 0,C 180,E1 -15930,E2 -15930} C_VEL
LIN {X 0,Y 303.577,Z 555.214,A -85,B 0,C 180,E1 -15932.654,E2 -15932.654} C_VEL
LIN {X 0,Y 303.683,Z 553.016,A -85,B 0,C 180,E1 -15935.311,E2 -15935.311} C_VEL
LIN {X 0,Y 303.941,Z 550.33,A -85,B 0,C 180,E1 -15937.306,E2 -15937.306} C_VEL
LIN {X 0,Y 304.427,Z 546.625,A -85,B 0,C 180,E1 -15939.3,E2 -15939.3} C_VEL
LIN {X 0,Y 305.17,Z 541.8,A -85,B 0,C 180,E1 -15941.289,E2 -15941.289} C_VEL
LIN {X 0,Y 306.165,Z 535.706,A -85,B 0,C 180,E1 -15943.27,E2 -15943.27} C_VEL
LIN {X 0,Y 307.359,Z 529.537,A -85,B 0,C 180,E1 -15944.906,E2 -15944.906} C_VEL
LIN {X 0,Y 308.618,Z 522.236,A -85,B 0,C 180,E1 -15946.514,E2 -15946.514} C_VEL
LIN {X 0,Y 309.951,Z 514.123,A -85,B 0,C 180,E1 -15947.995,E2 -15947.995} C_VEL
LIN {X 0,Y 311.329,Z 505.647,A -85,B 0,C 180,E1 -15949.278,E2 -15949.278} C_VEL
LIN {X 0,Y 312.871,Z 495.305,A -85,B 0,C 180,E1 -15950.547,E2 -15950.547} C_VEL
LIN {X 0,Y 314.238,Z 485.82,A -85,B 0,C 180,E1 -15951.483,E2 -15951.483} C_VEL
LIN {X 0,Y 315.308,Z 476.058,A -85,B 0,C 180,E1 -15952.267,E2 -15952.267} C_VEL
LIN {X 0,Y 316.387,Z 464.471,A -85,B 0,C 180,E1 -15952.962,E2 -15952.962} C_VEL
LIN {X 0,Y 317.232,Z 453.616,A -85,B 0,C 180,E1 -15953.415,E2 -15953.415} C_VEL
LIN {X 0,Y 317.791,Z 435.632,A -85,B 0,C 180,E1 -15953.896,E2 -15953.896} C_VEL
LIN {X 0,Y 319.189,Z 383.184,A -85,B 0,C 180,E1 -15955.12,E2 -15955.12} C_VEL
LIN {X 0,Y 315.512,Z 361.536,A -85,B 0,C 180,E1 -15956.044,E2 -15956.044} C_VEL
LIN {X 0,Y 313.584,Z 352.983,A -85,B 0,C 180,E1 -15956.466,E2 -15956.466} C_VEL
LIN {X 0,Y 309.644,Z 343.402,A -85,B 0,C 180,E1 -15957.19,E2 -15957.19} C_VEL
LIN {X 0,Y 308.251,Z 336.776,A -85,B 0,C 180,E1 -15959.25,E2 -15959.25} C_VEL
LIN {X 0,Y 305.943,Z 326.791,A -85,B 0,C 180,E1 -15962.671,E2 -15962.671} C_VEL
LIN {X 0,Y 305.511,Z 324.952,A -85,B 0,C 180,E1 -15963.462,E2 -15963.462} C_VEL
LIN {X 0,Y 305.473,Z 324.926,A -85,B 0,C 180,E1 -15966.74,E2 -15966.74} C_VEL
LIN {X 0,Y 305.452,Z 324.924,A -85,B 0,C 180,E1 -15970.6,E2 -15970.6} C_VEL
LIN {X 0,Y 305.423,Z 324.939,A -85,B 0,C 180,E1 -15973.655,E2 -15973.655} C_VEL
LIN {X 0,Y 305.453,Z 324.937,A -85,B 0,C 180,E1 -15977.415,E2 -15977.415} C_VEL
LIN {X 0,Y 305.466,Z 324.93,A -85,B 0,C 180,E1 -15981.597,E2 -15981.597} C_VEL
LIN {X 0,Y 305.461,Z 324.927,A -85,B 0,C 180,E1 -15984.887,E2 -15984.887} C_VEL
LIN {X 0,Y 305.449,Z 324.93,A -85,B 0,C 180,E1 -15988.356,E2 -15988.356} C_VEL
LIN {X 0,Y 305.512,Z 324.927,A -85,B 0,C 180,E1 -15991.113,E2 -15991.113} C_VEL
LIN {X 0,Y 305.571,Z 324.918,A -85,B 0,C 180,E1 -15994.088,E2 -15994.088} C_VEL
LIN {X 0,Y 305.501,Z 324.926,A -85,B 0,C 180,E1 -15998.403,E2 -15998.403} C_VEL
LIN {X 0,Y 305.59,Z 324.91,A -85,B 0,C 180,E1 -16001.218,E2 -16001.218} C_VEL
LIN {X 0,Y 305.649,Z 324.904,A -85,B 0,C 180,E1 -16005.349,E2 -16005.349} C_VEL
LIN {X 0,Y 305.64,Z 324.914,A -85,B 0,C 180,E1 -16009.4,E2 -16009.4} C_VEL
LIN {X 0,Y 305.815,Z 324.884,A -85,B 0,C 180,E1 -16012.075,E2 -16012.075} C_VEL
LIN {X 0,Y 305.691,Z 324.9,A -85,B 0,C 180,E1 -16014.724,E2 -16014.724} C_VEL
LIN {X 0,Y 305.959,Z 324.872,A -85,B 0,C 180,E1 -16018.684,E2 -16018.684} C_VEL
LIN {X 0,Y 305.959,Z 324.868,A -85,B 0,C 180,E1 -16021.317,E2 -16021.317} C_VEL
LIN {X 0,Y 305.854,Z 324.885,A -85,B 0,C 180,E1 -16026.598,E2 -16026.598} C_VEL
LIN {X 0,Y 305.737,Z 324.894,A -85,B 0,C 180,E1 -16029.26,E2 -16029.26} C_VEL
LIN {X 0,Y 305.59,Z 324.913,A -85,B 0,C 180,E1 -16033.296,E2 -16033.296} C_VEL
LIN {X 0,Y 305.595,Z 324.913,A -85,B 0,C 180,E1 -16036.02,E2 -16036.02} C_VEL
LIN {X 0,Y 305.561,Z 324.918,A -85,B 0,C 180,E1 -16039.436,E2 -16039.436} C_VEL
LIN {X 0,Y 305.487,Z 324.932,A -85,B 0,C 180,E1 -16043.04,E2 -16043.04} C_VEL
LIN {X 0,Y 305.502,Z 324.927,A -85,B 0,C 180,E1 -16046.209,E2 -16046.209} C_VEL
LIN {X 0,Y 305.485,Z 324.929,A -85,B 0,C 180,E1 -16049.046,E2 -16049.046} C_VEL
LIN {X 0,Y 305.443,Z 324.932,A -85,B 0,C 180,E1 -16051.953,E2 -16051.953} C_VEL
LIN {X 0,Y 305.511,Z 324.98,A -85,B 0,C 180,E1 -16054.963,E2 -16054.963} C_VEL
LIN {X 0,Y 307.126,Z 331.576,A -85,B 0,C 180,E1 -16057.329,E2 -16057.329} C_VEL
LIN {X 0,Y 308.232,Z 336.094,A -85,B 0,C 180,E1 -16058.728,E2 -16058.728} C_VEL
LIN {X 0,Y 315.858,Z 353.782,A -85,B 0,C 180,E1 -16060.03,E2 -16060.03} C_VEL
LIN {X 0,Y 317.226,Z 358.462,A -85,B 0,C 180,E1 -16060.289,E2 -16060.289} C_VEL
LIN {X 0,Y 319.482,Z 370.626,A -85,B 0,C 180,E1 -16060.826,E2 -16060.826} C_VEL
LIN {X 0,Y 317.376,Z 442.389,A -85,B 0,C 180,E1 -16062.525,E2 -16062.525} C_VEL
LIN {X 0,Y 316.803,Z 452.166,A -85,B 0,C 180,E1 -16062.881,E2 -16062.881} C_VEL
LIN {X 0,Y 316.08,Z 462.742,A -85,B 0,C 180,E1 -16063.447,E2 -16063.447} C_VEL
LIN {X 0,Y 315.108,Z 472.582,A -85,B 0,C 180,E1 -16064.133,E2 -16064.133} C_VEL
LIN {X 0,Y 314.047,Z 481.864,A -85,B 0,C 180,E1 -16064.95,E2 -16064.95} C_VEL
LIN {X 0,Y 312.592,Z 492.353,A -85,B 0,C 180,E1 -16066.111,E2 -16066.111} C_VEL
LIN {X 0,Y 311.181,Z 501.44,A -85,B 0,C 180,E1 -16067.348,E2 -16067.348} C_VEL
LIN {X 0,Y 309.594,Z 510.367,A -85,B 0,C 180,E1 -16068.828,E2 -16068.828} C_VEL
LIN {X 0,Y 308.3,Z 517.85,A -85,B 0,C 180,E1 -16070.336,E2 -16070.336} C_VEL
LIN {X 0,Y 307.175,Z 524.155,A -85,B 0,C 180,E1 -16071.848,E2 -16071.848} C_VEL
LIN {X 0,Y 305.946,Z 530.797,A -85,B 0,C 180,E1 -16073.811,E2 -16073.811} C_VEL
LIN {X 0,Y 305.174,Z 535.545,A -85,B 0,C 180,E1 -16075.535,E2 -16075.535} C_VEL
LIN {X 0,Y 304.559,Z 539.221,A -85,B 0,C 180,E1 -16077.161,E2 -16077.161} C_VEL
LIN {X 0,Y 303.966,Z 543.036,A -85,B 0,C 180,E1 -16079.425,E2 -16079.425} C_VEL
LIN {X 0,Y 303.564,Z 545.521,A -85,B 0,C 180,E1 -16081.614,E2 -16081.614} C_VEL
LIN {X 0,Y 303.278,Z 546.914,A -85,B 0,C 180,E1 -16083.877,E2 -16083.877} C_VEL
LIN {X 0,Y 303.216,Z 547.257,A -85,B 0,C 180,E1 -16085.342,E2 -16085.342} C_VEL
LIN {X 0,Y 303.302,Z 546.353,A -85,B 0,C 180,E1 -16088.238,E2 -16088.238} C_VEL
LIN {X 0,Y 303.422,Z 545.298,A -85,B 0,C 180,E1 -16089.67,E2 -16089.67} C_VEL
LIN {X 0,Y 303.736,Z 543.029,A -85,B 0,C 180,E1 -16091.565,E2 -16091.565} C_VEL
LIN {X 0,Y 304.197,Z 539.063,A -85,B 0,C 180,E1 -16093.904,E2 -16093.904} C_VEL
LIN {X 0,Y 304.852,Z 533.698,A -85,B 0,C 180,E1 -16096.162,E2 -16096.162} C_VEL
LIN {X 0,Y 305.649,Z 527.96,A -85,B 0,C 180,E1 -16098.057,E2 -16098.057} C_VEL
LIN {X 0,Y 306.617,Z 521.263,A -85,B 0,C 180,E1 -16099.848,E2 -16099.848} C_VEL
LIN {X 0,Y 307.748,Z 513.912,A -85,B 0,C 180,E1 -16101.464,E2 -16101.464} C_VEL
LIN {X 0,Y 308.893,Z 505.604,A -85,B 0,C 180,E1 -16102.976,E2 -16102.976} C_VEL
LIN {X 0,Y 310.064,Z 497.445,A -85,B 0,C 180,E1 -16104.211,E2 -16104.211} C_VEL
LIN {X 0,Y 311.31,Z 487.303,A -85,B 0,C 180,E1 -16105.468,E2 -16105.468} C_VEL
LIN {X 0,Y 312.388,Z 477.488,A -85,B 0,C 180,E1 -16106.453,E2 -16106.453} C_VEL
LIN {X 0,Y 313.412,Z 467.202,A -85,B 0,C 180,E1 -16107.269,E2 -16107.269} C_VEL
LIN {X 0,Y 314.165,Z 456.619,A -85,B 0,C 180,E1 -16107.917,E2 -16107.917} C_VEL
LIN {X 0,Y 314.845,Z 445.288,A -85,B 0,C 180,E1 -16108.401,E2 -16108.401} C_VEL
LIN {X 0,Y 315.39,Z 427.124,A -85,B 0,C 180,E1 -16108.879,E2 -16108.879} C_VEL
LIN {X 0,Y 316.702,Z 369.35,A -85,B 0,C 180,E1 -16110.219,E2 -16110.219} C_VEL
LIN {X 0,Y 312.838,Z 349.104,A -85,B 0,C 180,E1 -16111.019,E2 -16111.019} C_VEL
LIN {X 0,Y 308.189,Z 336.516,A -85,B 0,C 180,E1 -16111.74,E2 -16111.74} C_VEL
LIN {X 0,Y 307.624,Z 333.54,A -85,B 0,C 180,E1 -16112.619,E2 -16112.619} C_VEL
LIN {X 0,Y 305.752,Z 324.951,A -85,B 0,C 180,E1 -16115.689,E2 -16115.689} C_VEL
LIN {X 0,Y 305.757,Z 324.891,A -85,B 0,C 180,E1 -16118.743,E2 -16118.743} C_VEL
LIN {X 0,Y 305.591,Z 324.917,A -85,B 0,C 180,E1 -16123.296,E2 -16123.296} C_VEL
LIN {X 0,Y 305.596,Z 324.915,A -85,B 0,C 180,E1 -16126.02,E2 -16126.02} C_VEL
LIN {X 0,Y 305.562,Z 324.914,A -85,B 0,C 180,E1 -16129.436,E2 -16129.436} C_VEL
LIN {X 0,Y 305.488,Z 324.922,A -85,B 0,C 180,E1 -16133.039,E2 -16133.039} C_VEL
LIN {X 0,Y 305.549,Z 324.924,A -85,B 0,C 180,E1 -16136.227,E2 -16136.227} C_VEL
LIN {X 0,Y 305.489,Z 324.921,A -85,B 0,C 180,E1 -16139.047,E2 -16139.047} C_VEL
LIN {X 0,Y 305.444,Z 324.934,A -85,B 0,C 180,E1 -16141.952,E2 -16141.952} C_VEL
LIN {X 0,Y 305.464,Z 324.919,A -85,B 0,C 180,E1 -16145.113,E2 -16145.113} C_VEL
LIN {X 0,Y 305.468,Z 324.932,A -85,B 0,C 180,E1 -16148.533,E2 -16148.533} C_VEL
LIN {X 0,Y 305.461,Z 324.918,A -85,B 0,C 180,E1 -16152.587,E2 -16152.587} C_VEL
LIN {X 0,Y 305.424,Z 324.938,A -85,B 0,C 180,E1 -16155.925,E2 -16155.925} C_VEL
LIN {X 0,Y 304.778,Z 325.019,A -85,B 0,C 180,E1 -16157.025,E2 -16157.025} C_VEL
LIN {X 0,Y 301.917,Z 325.362,A -85,B 0,C 180,E1 -16158.815,E2 -16158.815} C_VEL
LIN {X 0,Y 299.485,Z 325.654,A -85,B 0,C 180,E1 -16160.267,E2 -16160.267} C_VEL
LIN {X 0,Y 298.457,Z 325.784,A -85,B 0,C 180,E1 -16161.392,E2 -16161.392} C_VEL
LIN {X 0,Y 298.382,Z 325.795,A -85,B 0,C 180,E1 -16161.774,E2 -16161.774} C_VEL
LIN {X 0,Y 298.43,Z 325.811,A -85,B 0,C 180,E1 -16165.513,E2 -16165.513} C_VEL
LIN {X 0,Y 298.379,Z 325.8,A -85,B 0,C 180,E1 -16168.789,E2 -16168.789} C_VEL
LIN {X 0,Y 298.417,Z 325.783,A -85,B 0,C 180,E1 -16171.899,E2 -16171.899} C_VEL
LIN {X 0,Y 298.451,Z 325.805,A -85,B 0,C 180,E1 -16174.921,E2 -16174.921} C_VEL
LIN {X 0,Y 298.432,Z 325.794,A -85,B 0,C 180,E1 -16179.314,E2 -16179.314} C_VEL
LIN {X 0,Y 298.481,Z 325.763,A -85,B 0,C 180,E1 -16182.176,E2 -16182.176} C_VEL
LIN {X 0,Y 298.588,Z 325.777,A -85,B 0,C 180,E1 -16184.994,E2 -16184.994} C_VEL
LIN {X 0,Y 298.585,Z 325.79,A -85,B 0,C 180,E1 -16189.146,E2 -16189.146} C_VEL
LIN {X 0,Y 298.699,Z 325.749,A -85,B 0,C 180,E1 -16191.884,E2 -16191.884} C_VEL
LIN {X 0,Y 298.631,Z 325.753,A -85,B 0,C 180,E1 -16194.598,E2 -16194.598} C_VEL
LIN {X 0,Y 298.905,Z 325.75,A -85,B 0,C 180,E1 -16198.652,E2 -16198.652} C_VEL
LIN {X 0,Y 298.915,Z 325.741,A -85,B 0,C 180,E1 -16201.347,E2 -16201.347} C_VEL
LIN {X 0,Y 298.755,Z 325.749,A -85,B 0,C 180,E1 -16206.755,E2 -16206.755} C_VEL
LIN {X 0,Y 298.627,Z 325.788,A -85,B 0,C 180,E1 -16209.482,E2 -16209.482} C_VEL
LIN {X 0,Y 298.524,Z 325.778,A -85,B 0,C 180,E1 -16213.616,E2 -16213.616} C_VEL
LIN {X 0,Y 298.454,Z 325.789,A -85,B 0,C 180,E1 -16216.414,E2 -16216.414} C_VEL
LIN {X 0,Y 298.443,Z 325.808,A -85,B 0,C 180,E1 -16219.617,E2 -16219.617} C_VEL
LIN {X 0,Y 298.42,Z 325.79,A -85,B 0,C 180,E1 -16223.6,E2 -16223.6} C_VEL
LIN {X 0,Y 298.407,Z 325.81,A -85,B 0,C 180,E1 -16226.582,E2 -16226.582} C_VEL
LIN {X 0,Y 298.393,Z 325.807,A -85,B 0,C 180,E1 -16229.644,E2 -16229.644} C_VEL
LIN {X 0,Y 298.392,Z 325.807,A -85,B 0,C 180,E1 -16232.8,E2 -16232.8} C_VEL
LIN {X 0,Y 298.426,Z 325.802,A -85,B 0,C 180,E1 -16236.802,E2 -16236.802} C_VEL
LIN {X 0,Y 298.346,Z 325.819,A -85,B 0,C 180,E1 -16241.268,E2 -16241.268} C_VEL
LIN {X 0,Y 298.353,Z 325.819,A -85,B 0,C 180,E1 -16245.034,E2 -16245.034} C_VEL
LIN {X 0,Y 298.346,Z 325.819,A -85,B 0,C 180,E1 -16248.921,E2 -16248.921} C_VEL
LIN {X 0,Y 298.396,Z 325.814,A -85,B 0,C 180,E1 -16252.239,E2 -16252.239} C_VEL
LIN {X 0,Y 298.406,Z 325.808,A -85,B 0,C 180,E1 -16255.581,E2 -16255.581} C_VEL
LIN {X 0,Y 298.398,Z 325.961,A -85,B 0,C 180,E1 -16257.767,E2 -16257.767} C_VEL
LIN {X 0,Y 300.392,Z 335.142,A -85,B 0,C 180,E1 -16260.957,E2 -16260.957} C_VEL
LIN {X 0,Y 302.162,Z 343.944,A -85,B 0,C 180,E1 -16263.773,E2 -16263.773} C_VEL
LIN {X 0,Y 303.89,Z 348.903,A -85,B 0,C 180,E1 -16264.112,E2 -16264.112} C_VEL
LIN {X 0,Y 305.375,Z 355.485,A -85,B 0,C 180,E1 -16264.403,E2 -16264.403} C_VEL
LIN {X 0,Y 309.898,Z 383.114,A -85,B 0,C 180,E1 -16265.46,E2 -16265.46} C_VEL
LIN {X 0,Y 308.169,Z 450.322,A -85,B 0,C 180,E1 -16267.078,E2 -16267.078} C_VEL
LIN {X 0,Y 307.677,Z 460.42,A -85,B 0,C 180,E1 -16267.46,E2 -16267.46} C_VEL
LIN {X 0,Y 306.897,Z 470.213,A -85,B 0,C 180,E1 -16267.976,E2 -16267.976} C_VEL
LIN {X 0,Y 305.876,Z 481.407,A -85,B 0,C 180,E1 -16268.784,E2 -16268.784} C_VEL
LIN {X 0,Y 304.868,Z 490.348,A -85,B 0,C 180,E1 -16269.594,E2 -16269.594} C_VEL
LIN {X 0,Y 303.576,Z 500.448,A -85,B 0,C 180,E1 -16270.737,E2 -16270.737} C_VEL
LIN {X 0,Y 302.286,Z 509.893,A -85,B 0,C 180,E1 -16272.058,E2 -16272.058} C_VEL
LIN {X 0,Y 301.197,Z 517.96,A -85,B 0,C 180,E1 -16273.421,E2 -16273.421} C_VEL
LIN {X 0,Y 299.96,Z 526.02,A -85,B 0,C 180,E1 -16275.065,E2 -16275.065} C_VEL
LIN {X 0,Y 298.865,Z 532.844,A -85,B 0,C 180,E1 -16276.745,E2 -16276.745} C_VEL
LIN {X 0,Y 298.071,Z 538.546,A -85,B 0,C 180,E1 -16278.439,E2 -16278.439} C_VEL
LIN {X 0,Y 297.319,Z 544.064,A -85,B 0,C 180,E1 -16280.476,E2 -16280.476} C_VEL
LIN {X 0,Y 296.842,Z 548.388,A -85,B 0,C 180,E1 -16282.518,E2 -16282.518} C_VEL
LIN {X 0,Y 296.549,Z 551.636,A -85,B 0,C 180,E1 -16284.56,E2 -16284.56} C_VEL
LIN {X 0,Y 296.488,Z 553.267,A -85,B 0,C 180,E1 -16285.922,E2 -16285.922} C_VEL
LIN {X 0,Y 296.444,Z 555.226,A -85,B 0,C 180,E1 -16288.641,E2 -16288.641} C_VEL
LIN {X 0,Y 296.448,Z 555.542,A -85,B 0,C 180,E1 -16290,E2 -16290} C_VEL
LIN {X 0,Y 296.483,Z 555.136,A -85,B 0,C 180,E1 -16292.717,E2 -16292.717} C_VEL
LIN {X 0,Y 296.627,Z 552.692,A -85,B 0,C 180,E1 -16295.676,E2 -16295.676} C_VEL
LIN {X 0,Y 296.869,Z 550.321,A -85,B 0,C 180,E1 -16297.481,E2 -16297.481} C_VEL
LIN {X 0,Y 297.391,Z 546.645,A -85,B 0,C 180,E1 -16299.522,E2 -16299.522} C_VEL
LIN {X 0,Y 298.187,Z 541.851,A -85,B 0,C 180,E1 -16301.557,E2 -16301.557} C_VEL
LIN {X 0,Y 299.249,Z 535.79,A -85,B 0,C 180,E1 -16303.583,E2 -16303.583} C_VEL
LIN {X 0,Y 300.495,Z 529.657,A -85,B 0,C 180,E1 -16305.255,E2 -16305.255} C_VEL
LIN {X 0,Y 301.757,Z 522.664,A -85,B 0,C 180,E1 -16306.846,E2 -16306.846} C_VEL
LIN {X 0,Y 303.369,Z 513.316,A -85,B 0,C 180,E1 -16308.574,E2 -16308.574} C_VEL
LIN {X 0,Y 304.841,Z 504.696,A -85,B 0,C 180,E1 -16309.88,E2 -16309.88} C_VEL
LIN {X 0,Y 306.267,Z 495.661,A -85,B 0,C 180,E1 -16311.011,E2 -16311.011} C_VEL
LIN {X 0,Y 307.669,Z 486.306,A -85,B 0,C 180,E1 -16311.965,E2 -16311.965} C_VEL
LIN {X 0,Y 308.918,Z 475.536,A -85,B 0,C 180,E1 -16312.841,E2 -16312.841} C_VEL
LIN {X 0,Y 309.952,Z 464.644,A -85,B 0,C 180,E1 -16313.511,E2 -16313.511} C_VEL
LIN {X 0,Y 310.843,Z 453.961,A -85,B 0,C 180,E1 -16313.97,E2 -16313.97} C_VEL
LIN {X 0,Y 311.423,Z 436.328,A -85,B 0,C 180,E1 -16314.458,E2 -16314.458} C_VEL
LIN {X 0,Y 312.808,Z 383.373,A -85,B 0,C 180,E1 -16315.73,E2 -16315.73} C_VEL
LIN {X 0,Y 308.754,Z 359.883,A -85,B 0,C 180,E1 -16316.778,E2 -16316.778} C_VEL
LIN {X 0,Y 307.49,Z 355.183,A -85,B 0,C 180,E1 -16317.043,E2 -16317.043} C_VEL
LIN {X 0,Y 302.505,Z 343.469,A -85,B 0,C 180,E1 -16317.962,E2 -16317.962} C_VEL
LIN {X 0,Y 302.041,Z 341.443,A -85,B 0,C 180,E1 -16318.499,E2 -16318.499} C_VEL
LIN {X 0,Y 299.954,Z 332.059,A -85,B 0,C 180,E1 -16321.734,E2 -16321.734} C_VEL
LIN {X 0,Y 298.429,Z 325.894,A -85,B 0,C 180,E1 -16324.059,E2 -16324.059} C_VEL
LIN {X 0,Y 298.412,Z 325.81,A -85,B 0,C 180,E1 -16327.758,E2 -16327.758} C_VEL
LIN {X 0,Y 298.381,Z 325.809,A -85,B 0,C 180,E1 -16331.262,E2 -16331.262} C_VEL
LIN {X 0,Y 298.352,Z 325.821,A -85,B 0,C 180,E1 -16335.035,E2 -16335.035} C_VEL
LIN {X 0,Y 298.383,Z 325.811,A -85,B 0,C 180,E1 -16338.739,E2 -16338.739} C_VEL
LIN {X 0,Y 298.407,Z 325.812,A -85,B 0,C 180,E1 -16342.241,E2 -16342.241} C_VEL
LIN {X 0,Y 298.407,Z 325.807,A -85,B 0,C 180,E1 -16345.581,E2 -16345.581} C_VEL
LIN {X 0,Y 298.391,Z 325.809,A -85,B 0,C 180,E1 -16348.791,E2 -16348.791} C_VEL
LIN {X 0,Y 298.458,Z 325.802,A -85,B 0,C 180,E1 -16351.904,E2 -16351.904} C_VEL
LIN {X 0,Y 298.485,Z 325.805,A -85,B 0,C 180,E1 -16354.924,E2 -16354.924} C_VEL
LIN {X 0,Y 298.45,Z 325.809,A -85,B 0,C 180,E1 -16359.316,E2 -16359.316} C_VEL
LIN {X 0,Y 298.538,Z 325.789,A -85,B 0,C 180,E1 -16362.18,E2 -16362.18} C_VEL
LIN {X 0,Y 298.594,Z 325.787,A -85,B 0,C 180,E1 -16364.995,E2 -16364.995} C_VEL
LIN {X 0,Y 298.595,Z 325.79,A -85,B 0,C 180,E1 -16369.147,E2 -16369.147} C_VEL
LIN {X 0,Y 298.761,Z 325.76,A -85,B 0,C 180,E1 -16371.886,E2 -16371.886} C_VEL
LIN {X 0,Y 298.662,Z 325.776,A -85,B 0,C 180,E1 -16374.599,E2 -16374.599} C_VEL
LIN {X 0,Y 298.925,Z 325.748,A -85,B 0,C 180,E1 -16378.653,E2 -16378.653} C_VEL
LIN {X 0,Y 298.925,Z 325.744,A -85,B 0,C 180,E1 -16381.348,E2 -16381.348} C_VEL
LIN {X 0,Y 298.8,Z 325.765,A -85,B 0,C 180,E1 -16386.754,E2 -16386.754} C_VEL
LIN {X 0,Y 298.682,Z 325.774,A -85,B 0,C 180,E1 -16389.481,E2 -16389.481} C_VEL
LIN {X 0,Y 298.553,Z 325.793,A -85,B 0,C 180,E1 -16393.616,E2 -16393.616} C_VEL
LIN {X 0,Y 298.55,Z 325.791,A -85,B 0,C 180,E1 -16396.409,E2 -16396.409} C_VEL
LIN {X 0,Y 298.499,Z 325.798,A -85,B 0,C 180,E1 -16399.648,E2 -16399.648} C_VEL
LIN {X 0,Y 298.425,Z 325.813,A -85,B 0,C 180,E1 -16403.601,E2 -16403.601} C_VEL
LIN {X 0,Y 298.455,Z 325.8,A -85,B 0,C 180,E1 -16406.578,E2 -16406.578} C_VEL
LIN {X 0,Y 298.415,Z 325.814,A -85,B 0,C 180,E1 -16409.642,E2 -16409.642} C_VEL
LIN {X 0,Y 298.449,Z 325.828,A -85,B 0,C 180,E1 -16414.21,E2 -16414.21} C_VEL
LIN {X 0,Y 298.524,Z 326.244,A -85,B 0,C 180,E1 -16414.514,E2 -16414.514} C_VEL
LIN {X 0,Y 300.93,Z 335.902,A -85,B 0,C 180,E1 -16417.864,E2 -16417.864} C_VEL
LIN {X 0,Y 302.834,Z 340.125,A -85,B 0,C 180,E1 -16418.269,E2 -16418.269} C_VEL
LIN {X 0,Y 310.237,Z 357.293,A -85,B 0,C 180,E1 -16419.552,E2 -16419.552} C_VEL
LIN {X 0,Y 311.344,Z 361.407,A -85,B 0,C 180,E1 -16419.778,E2 -16419.778} C_VEL
LIN {X 0,Y 313.202,Z 371.984,A -85,B 0,C 180,E1 -16420.249,E2 -16420.249} C_VEL
LIN {X 0,Y 311.047,Z 442.098,A -85,B 0,C 180,E1 -16421.941,E2 -16421.941} C_VEL
LIN {X 0,Y 310.489,Z 451.645,A -85,B 0,C 180,E1 -16422.287,E2 -16422.287} C_VEL
LIN {X 0,Y 309.691,Z 462.074,A -85,B 0,C 180,E1 -16422.837,E2 -16422.837} C_VEL
LIN {X 0,Y 308.655,Z 472.597,A -85,B 0,C 180,E1 -16423.584,E2 -16423.584} C_VEL
LIN {X 0,Y 307.529,Z 481.981,A -85,B 0,C 180,E1 -16424.426,E2 -16424.426} C_VEL
LIN {X 0,Y 305.927,Z 492.928,A -85,B 0,C 180,E1 -16425.671,E2 -16425.671} C_VEL
LIN {X 0,Y 304.543,Z 501.536,A -85,B 0,C 180,E1 -16426.87,E2 -16426.87} C_VEL
LIN {X 0,Y 303.093,Z 509.511,A -85,B 0,C 180,E1 -16428.196,E2 -16428.196} C_VEL
LIN {X 0,Y 301.535,Z 517.918,A -85,B 0,C 180,E1 -16429.912,E2 -16429.912} C_VEL
LIN {X 0,Y 300.197,Z 524.924,A -85,B 0,C 180,E1 -16431.655,E2 -16431.655} C_VEL
LIN {X 0,Y 299.037,Z 530.891,A -85,B 0,C 180,E1 -16433.466,E2 -16433.466} C_VEL
LIN {X 0,Y 298.423,Z 534.527,A -85,B 0,C 180,E1 -16434.761,E2 -16434.761} C_VEL
LIN {X 0,Y 297.494,Z 539.673,A -85,B 0,C 180,E1 -16437.088,E2 -16437.088} C_VEL
LIN {X 0,Y 297.042,Z 542.283,A -85,B 0,C 180,E1 -16438.633,E2 -16438.633} C_VEL
LIN {X 0,Y 296.534,Z 545.493,A -85,B 0,C 180,E1 -16441.273,E2 -16441.273} C_VEL
LIN {X 0,Y 296.257,Z 546.84,A -85,B 0,C 180,E1 -16443.21,E2 -16443.21} C_VEL
LIN {X 0,Y 296.166,Z 547.229,A -85,B 0,C 180,E1 -16444.714,E2 -16444.714} C_VEL
LIN {X 0,Y 296.154,Z 546.831,A -85,B 0,C 180,E1 -16447.685,E2 -16447.685} C_VEL
LIN {X 0,Y 296.265,Z 545.797,A -85,B 0,C 180,E1 -16449.156,E2 -16449.156} C_VEL
LIN {X 0,Y 296.607,Z 543.42,A -85,B 0,C 180,E1 -16451.404,E2 -16451.404} C_VEL
LIN {X 0,Y 297.009,Z 540.111,A -85,B 0,C 180,E1 -16453.504,E2 -16453.504} C_VEL
LIN {X 0,Y 297.556,Z 535.78,A -85,B 0,C 180,E1 -16455.554,E2 -16455.554} C_VEL
LIN {X 0,Y 298.563,Z 528.67,A -85,B 0,C 180,E1 -16458.114,E2 -16458.114} C_VEL
LIN {X 0,Y 299.649,Z 521.493,A -85,B 0,C 180,E1 -16460.089,E2 -16460.089} C_VEL
LIN {X 0,Y 300.713,Z 514.881,A -85,B 0,C 180,E1 -16461.601,E2 -16461.601} C_VEL
LIN {X 0,Y 302.037,Z 505.677,A -85,B 0,C 180,E1 -16463.319,E2 -16463.319} C_VEL
LIN {X 0,Y 303.333,Z 496.753,A -85,B 0,C 180,E1 -16464.683,E2 -16464.683} C_VEL
LIN {X 0,Y 304.553,Z 487.247,A -85,B 0,C 180,E1 -16465.876,E2 -16465.876} C_VEL
LIN {X 0,Y 305.665,Z 477.515,A -85,B 0,C 180,E1 -16466.87,E2 -16466.87} C_VEL
LIN {X 0,Y 306.719,Z 467.211,A -85,B 0,C 180,E1 -16467.702,E2 -16467.702} C_VEL
LIN {X 0,Y 307.476,Z 456.622,A -85,B 0,C 180,E1 -16468.363,E2 -16468.363} C_VEL
LIN {X 0,Y 308.183,Z 446.063,A -85,B 0,C 180,E1 -16468.828,E2 -16468.828} C_VEL
LIN {X 0,Y 308.717,Z 429.705,A -85,B 0,C 180,E1 -16469.279,E2 -16469.279} C_VEL
LIN {X 0,Y 310.15,Z 370.463,A -85,B 0,C 180,E1 -16470.679,E2 -16470.679} C_VEL
LIN {X 0,Y 306.601,Z 351.719,A -85,B 0,C 180,E1 -16471.437,E2 -16471.437} C_VEL
LIN {X 0,Y 301.027,Z 336.566,A -85,B 0,C 180,E1 -16472.332,E2 -16472.332} C_VEL
LIN {X 0,Y 300.279,Z 333.315,A -85,B 0,C 180,E1 -16473.355,E2 -16473.355} C_VEL
LIN {X 0,Y 298.765,Z 325.825,A -85,B 0,C 180,E1 -16476.119,E2 -16476.119} C_VEL
LIN {X 0,Y 298.627,Z 325.785,A -85,B 0,C 180,E1 -16479.482,E2 -16479.482} C_VEL
LIN {X 0,Y 298.554,Z 325.796,A -85,B 0,C 180,E1 -16483.615,E2 -16483.615} C_VEL
LIN {X 0,Y 298.551,Z 325.796,A -85,B 0,C 180,E1 -16486.409,E2 -16486.409} C_VEL
LIN {X 0,Y 298.5,Z 325.795,A -85,B 0,C 180,E1 -16489.647,E2 -16489.647} C_VEL
LIN {X 0,Y 298.431,Z 325.801,A -85,B 0,C 180,E1 -16493.6,E2 -16493.6} C_VEL
LIN {X 0,Y 298.491,Z 325.802,A -85,B 0,C 180,E1 -16496.574,E2 -16496.574} C_VEL
LIN {X 0,Y 298.418,Z 325.809,A -85,B 0,C 180,E1 -16499.641,E2 -16499.641} C_VEL
LIN {X 0,Y 298.396,Z 325.811,A -85,B 0,C 180,E1 -16502.8,E2 -16502.8} C_VEL
LIN {X 0,Y 298.466,Z 325.803,A -85,B 0,C 180,E1 -16506.812,E2 -16506.812} C_VEL
LIN {X 0,Y 298.389,Z 325.797,A -85,B 0,C 180,E1 -16511.088,E2 -16511.088} C_VEL
LIN {X 0,Y 298.39,Z 325.815,A -85,B 0,C 180,E1 -16515.041,E2 -16515.041} C_VEL
LIN {X 0,Y 298.388,Z 325.797,A -85,B 0,C 180,E1 -16518.913,E2 -16518.913} C_VEL
LIN {X 0,Y 298.382,Z 325.795,A -85,B 0,C 180,E1 -16521.774,E2 -16521.774} C_VEL
LIN {X 0,Y 297.724,Z 325.887,A -85,B 0,C 180,E1 -16522.901,E2 -16522.901} C_VEL
LIN {X 0,Y 294.835,Z 326.258,A -85,B 0,C 180,E1 -16524.734,E2 -16524.734} C_VEL
LIN {X 0,Y 292.405,Z 326.559,A -85,B 0,C 180,E1 -16526.223,E2 -16526.223} C_VEL
LIN {X 0,Y 291.408,Z 326.678,A -85,B 0,C 180,E1 -16527.377,E2 -16527.377} C_VEL
LIN {X 0,Y 291.352,Z 326.68,A -85,B 0,C 180,E1 -16527.768,E2 -16527.768} C_VEL
LIN {X 0,Y 291.347,Z 326.657,A -85,B 0,C 180,E1 -16531.154,E2 -16531.154} C_VEL
LIN {X 0,Y 291.378,Z 326.683,A -85,B 0,C 180,E1 -16534.268,E2 -16534.268} C_VEL
LIN {X 0,Y 291.374,Z 326.685,A -85,B 0,C 180,E1 -16537.299,E2 -16537.299} C_VEL
LIN {X 0,Y 291.441,Z 326.653,A -85,B 0,C 180,E1 -16540.269,E2 -16540.269} C_VEL
LIN {X 0,Y 291.517,Z 326.654,A -85,B 0,C 180,E1 -16544.653,E2 -16544.653} C_VEL
LIN {X 0,Y 291.531,Z 326.668,A -85,B 0,C 180,E1 -16548.88,E2 -16548.88} C_VEL
LIN {X 0,Y 291.653,Z 326.628,A -85,B 0,C 180,E1 -16551.687,E2 -16551.687} C_VEL
LIN {X 0,Y 291.601,Z 326.626,A -85,B 0,C 180,E1 -16554.467,E2 -16554.467} C_VEL
LIN {X 0,Y 291.873,Z 326.627,A -85,B 0,C 180,E1 -16558.62,E2 -16558.62} C_VEL
LIN {X 0,Y 291.881,Z 326.617,A -85,B 0,C 180,E1 -16561.379,E2 -16561.379} C_VEL
LIN {X 0,Y 291.706,Z 326.628,A -85,B 0,C 180,E1 -16566.919,E2 -16566.919} C_VEL
LIN {X 0,Y 291.57,Z 326.665,A -85,B 0,C 180,E1 -16569.714,E2 -16569.714} C_VEL
LIN {X 0,Y 291.483,Z 326.651,A -85,B 0,C 180,E1 -16573.952,E2 -16573.952} C_VEL
LIN {X 0,Y 291.406,Z 326.673,A -85,B 0,C 180,E1 -16576.822,E2 -16576.822} C_VEL
LIN {X 0,Y 291.392,Z 326.689,A -85,B 0,C 180,E1 -16579.841,E2 -16579.841} C_VEL
LIN {X 0,Y 291.359,Z 326.669,A -85,B 0,C 180,E1 -16584.208,E2 -16584.208} C_VEL
LIN {X 0,Y 291.353,Z 326.692,A -85,B 0,C 180,E1 -16587.278,E2 -16587.278} C_VEL
LIN {X 0,Y 291.318,Z 326.684,A -85,B 0,C 180,E1 -16590.439,E2 -16590.439} C_VEL
LIN {X 0,Y 291.343,Z 326.695,A -85,B 0,C 180,E1 -16593.698,E2 -16593.698} C_VEL
LIN {X 0,Y 291.352,Z 326.681,A -85,B 0,C 180,E1 -16597.247,E2 -16597.247} C_VEL
LIN {X 0,Y 291.293,Z 326.695,A -85,B 0,C 180,E1 -16601.588,E2 -16601.588} C_VEL
LIN {X 0,Y 291.28,Z 326.7,A -85,B 0,C 180,E1 -16605.596,E2 -16605.596} C_VEL
LIN {X 0,Y 291.298,Z 326.696,A -85,B 0,C 180,E1 -16609.351,E2 -16609.351} C_VEL
LIN {X 0,Y 291.388,Z 326.691,A -85,B 0,C 180,E1 -16612.916,E2 -16612.916} C_VEL
LIN {X 0,Y 291.371,Z 326.736,A -85,B 0,C 180,E1 -16617.237,E2 -16617.237} C_VEL
LIN {X 0,Y 292.008,Z 329.835,A -85,B 0,C 180,E1 -16618.434,E2 -16618.434} C_VEL
LIN {X 0,Y 293.837,Z 338.488,A -85,B 0,C 180,E1 -16621.421,E2 -16621.421} C_VEL
LIN {X 0,Y 294.99,Z 344.036,A -85,B 0,C 180,E1 -16623.188,E2 -16623.188} C_VEL
LIN {X 0,Y 298.321,Z 353.567,A -85,B 0,C 180,E1 -16623.77,E2 -16623.77} C_VEL
LIN {X 0,Y 303.276,Z 383.354,A -85,B 0,C 180,E1 -16624.959,E2 -16624.959} C_VEL
LIN {X 0,Y 301.565,Z 449.669,A -85,B 0,C 180,E1 -16626.59,E2 -16626.59} C_VEL
LIN {X 0,Y 301.03,Z 459.994,A -85,B 0,C 180,E1 -16626.98,E2 -16626.98} C_VEL
LIN {X 0,Y 300.34,Z 469.277,A -85,B 0,C 180,E1 -16627.469,E2 -16627.469} C_VEL
LIN {X 0,Y 299.21,Z 480.65,A -85,B 0,C 180,E1 -16628.288,E2 -16628.288} C_VEL
LIN {X 0,Y 298.006,Z 491.232,A -85,B 0,C 180,E1 -16629.283,E2 -16629.283} C_VEL
LIN {X 0,Y 296.662,Z 501.156,A -85,B 0,C 180,E1 -16630.45,E2 -16630.45} C_VEL
LIN {X 0,Y 295.506,Z 509.436,A -85,B 0,C 180,E1 -16631.632,E2 -16631.632} C_VEL
LIN {X 0,Y 294.301,Z 517.945,A -85,B 0,C 180,E1 -16633.1,E2 -16633.1} C_VEL
LIN {X 0,Y 293.054,Z 525.673,A -85,B 0,C 180,E1 -16634.704,E2 -16634.704} C_VEL
LIN {X 0,Y 291.94,Z 532.542,A -85,B 0,C 180,E1 -16636.425,E2 -16636.425} C_VEL
LIN {X 0,Y 291.06,Z 538.281,A -85,B 0,C 180,E1 -16638.156,E2 -16638.156} C_VEL
LIN {X 0,Y 290.296,Z 543.834,A -85,B 0,C 180,E1 -16640.243,E2 -16640.243} C_VEL
LIN {X 0,Y 289.784,Z 548.19,A -85,B 0,C 180,E1 -16642.334,E2 -16642.334} C_VEL
LIN {X 0,Y 289.473,Z 551.566,A -85,B 0,C 180,E1 -16644.51,E2 -16644.51} C_VEL
LIN {X 0,Y 289.394,Z 553.099,A -85,B 0,C 180,E1 -16645.822,E2 -16645.822} C_VEL
LIN {X 0,Y 289.368,Z 555.114,A -85,B 0,C 180,E1 -16648.608,E2 -16648.608} C_VEL
LIN {X 0,Y 289.368,Z 555.398,A -85,B 0,C 180,E1 -16651.392,E2 -16651.392} C_VEL
LIN {X 0,Y 289.391,Z 555.058,A -85,B 0,C 180,E1 -16652.784,E2 -16652.784} C_VEL
LIN {X 0,Y 289.513,Z 552.943,A -85,B 0,C 180,E1 -16655.572,E2 -16655.572} C_VEL
LIN {X 0,Y 289.825,Z 550.313,A -85,B 0,C 180,E1 -16657.664,E2 -16657.664} C_VEL
LIN {X 0,Y 290.366,Z 546.666,A -85,B 0,C 180,E1 -16659.754,E2 -16659.754} C_VEL
LIN {X 0,Y 291.215,Z 541.902,A -85,B 0,C 180,E1 -16661.837,E2 -16661.837} C_VEL
LIN {X 0,Y 292.351,Z 535.873,A -85,B 0,C 180,E1 -16663.91,E2 -16663.91} C_VEL
LIN {X 0,Y 293.648,Z 529.78,A -85,B 0,C 180,E1 -16665.62,E2 -16665.62} C_VEL
LIN {X 0,Y 295.049,Z 522.065,A -85,B 0,C 180,E1 -16667.405,E2 -16667.405} C_VEL
LIN {X 0,Y 296.639,Z 513.564,A -85,B 0,C 180,E1 -16669.012,E2 -16669.012} C_VEL
LIN {X 0,Y 298.185,Z 505.032,A -85,B 0,C 180,E1 -16670.343,E2 -16670.343} C_VEL
LIN {X 0,Y 299.682,Z 496.106,A -85,B 0,C 180,E1 -16671.495,E2 -16671.495} C_VEL
LIN {X 0,Y 301.13,Z 486.884,A -85,B 0,C 180,E1 -16672.468,E2 -16672.468} C_VEL
LIN {X 0,Y 302.558,Z 475.113,A -85,B 0,C 180,E1 -16673.44,E2 -16673.44} C_VEL
LIN {X 0,Y 303.628,Z 464.106,A -85,B 0,C 180,E1 -16674.122,E2 -16674.122} C_VEL
LIN {X 0,Y 304.539,Z 453.551,A -85,B 0,C 180,E1 -16674.576,E2 -16674.576} C_VEL
LIN {X 0,Y 305.134,Z 435.757,A -85,B 0,C 180,E1 -16675.077,E2 -16675.077} C_VEL
LIN {X 0,Y 306.591,Z 384.602,A -85,B 0,C 180,E1 -16676.325,E2 -16676.325} C_VEL
LIN {X 0,Y 302.568,Z 361.006,A -85,B 0,C 180,E1 -16677.412,E2 -16677.412} C_VEL
LIN {X 0,Y 300.959,Z 356.259,A -85,B 0,C 180,E1 -16677.727,E2 -16677.727} C_VEL
LIN {X 0,Y 295.316,Z 343.385,A -85,B 0,C 180,E1 -16678.802,E2 -16678.802} C_VEL
LIN {X 0,Y 294.907,Z 341.682,A -85,B 0,C 180,E1 -16679.245,E2 -16679.245} C_VEL
LIN {X 0,Y 292.669,Z 331.713,A -85,B 0,C 180,E1 -16682.811,E2 -16682.811} C_VEL
LIN {X 0,Y 291.394,Z 326.767,A -85,B 0,C 180,E1 -16684.781,E2 -16684.781} C_VEL
LIN {X 0,Y 291.374,Z 326.682,A -85,B 0,C 180,E1 -16687.254,E2 -16687.254} C_VEL
LIN {X 0,Y 291.33,Z 326.683,A -85,B 0,C 180,E1 -16690.643,E2 -16690.643} C_VEL
LIN {X 0,Y 291.288,Z 326.701,A -85,B 0,C 180,E1 -16694.402,E2 -16694.402} C_VEL
LIN {X 0,Y 291.325,Z 326.69,A -85,B 0,C 180,E1 -16698.405,E2 -16698.405} C_VEL
LIN {X 0,Y 291.346,Z 326.689,A -85,B 0,C 180,E1 -16701.158,E2 -16701.158} C_VEL
LIN {X 0,Y 291.36,Z 326.684,A -85,B 0,C 180,E1 -16704.626,E2 -16704.626} C_VEL
LIN {X 0,Y 291.37,Z 326.685,A -85,B 0,C 180,E1 -16707.951,E2 -16707.951} C_VEL
LIN {X 0,Y 291.377,Z 326.687,A -85,B 0,C 180,E1 -16711.158,E2 -16711.158} C_VEL
LIN {X 0,Y 291.416,Z 326.683,A -85,B 0,C 180,E1 -16714.272,E2 -16714.272} C_VEL
LIN {X 0,Y 291.381,Z 326.68,A -85,B 0,C 180,E1 -16717.3,E2 -16717.3} C_VEL
LIN {X 0,Y 291.458,Z 326.677,A -85,B 0,C 180,E1 -16720.271,E2 -16720.271} C_VEL
LIN {X 0,Y 291.555,Z 326.665,A -85,B 0,C 180,E1 -16724.624,E2 -16724.624} C_VEL
LIN {X 0,Y 291.538,Z 326.668,A -85,B 0,C 180,E1 -16728.881,E2 -16728.881} C_VEL
LIN {X 0,Y 291.711,Z 326.637,A -85,B 0,C 180,E1 -16731.689,E2 -16731.689} C_VEL
LIN {X 0,Y 291.632,Z 326.653,A -85,B 0,C 180,E1 -16734.469,E2 -16734.469} C_VEL
LIN {X 0,Y 291.891,Z 326.625,A -85,B 0,C 180,E1 -16738.621,E2 -16738.621} C_VEL
LIN {X 0,Y 291.891,Z 326.62,A -85,B 0,C 180,E1 -16741.38,E2 -16741.38} C_VEL
LIN {X 0,Y 291.748,Z 326.645,A -85,B 0,C 180,E1 -16746.918,E2 -16746.918} C_VEL
LIN {X 0,Y 291.631,Z 326.654,A -85,B 0,C 180,E1 -16749.712,E2 -16749.712} C_VEL
LIN {X 0,Y 291.523,Z 326.672,A -85,B 0,C 180,E1 -16753.951,E2 -16753.951} C_VEL
LIN {X 0,Y 291.487,Z 326.673,A -85,B 0,C 180,E1 -16756.818,E2 -16756.818} C_VEL
LIN {X 0,Y 291.452,Z 326.677,A -85,B 0,C 180,E1 -16759.875,E2 -16759.875} C_VEL
LIN {X 0,Y 291.372,Z 326.688,A -85,B 0,C 180,E1 -16764.208,E2 -16764.208} C_VEL
LIN {X 0,Y 291.401,Z 326.673,A -85,B 0,C 180,E1 -16767.274,E2 -16767.274} C_VEL
LIN {X 0,Y 291.334,Z 326.689,A -85,B 0,C 180,E1 -16770.438,E2 -16770.438} C_VEL
LIN {X 0,Y 291.423,Z 326.779,A -85,B 0,C 180,E1 -16773.59,E2 -16773.59} C_VEL
LIN {X 0,Y 293.533,Z 335.221,A -85,B 0,C 180,E1 -16776.768,E2 -16776.768} C_VEL
LIN {X 0,Y 293.907,Z 336.511,A -85,B 0,C 180,E1 -16777.086,E2 -16777.086} C_VEL
LIN {X 0,Y 300.477,Z 350.603,A -85,B 0,C 180,E1 -16778.303,E2 -16778.303} C_VEL
LIN {X 0,Y 304.946,Z 361.763,A -85,B 0,C 180,E1 -16779.117,E2 -16779.117} C_VEL
LIN {X 0,Y 306.91,Z 372.394,A -85,B 0,C 180,E1 -16779.618,E2 -16779.618} C_VEL
LIN {X 0,Y 305.261,Z 429.06,A -85,B 0,C 180,E1 -16780.999,E2 -16780.999} C_VEL
LIN {X 0,Y 304.514,Z 446.957,A -85,B 0,C 180,E1 -16781.496,E2 -16781.496} C_VEL
LIN {X 0,Y 303.389,Z 461.463,A -85,B 0,C 180,E1 -16782.205,E2 -16782.205} C_VEL
LIN {X 0,Y 302.22,Z 472.814,A -85,B 0,C 180,E1 -16783.024,E2 -16783.024} C_VEL
LIN {X 0,Y 300.936,Z 482.942,A -85,B 0,C 180,E1 -16783.966,E2 -16783.966} C_VEL
LIN {X 0,Y 299.477,Z 492.534,A -85,B 0,C 180,E1 -16785.073,E2 -16785.073} C_VEL
LIN {X 0,Y 297.929,Z 501.683,A -85,B 0,C 180,E1 -16786.37,E2 -16786.37} C_VEL
LIN {X 0,Y 296.551,Z 508.986,A -85,B 0,C 180,E1 -16787.594,E2 -16787.594} C_VEL
LIN {X 0,Y 294.762,Z 518.059,A -85,B 0,C 180,E1 -16789.48,E2 -16789.48} C_VEL
LIN {X 0,Y 293.528,Z 524.356,A -85,B 0,C 180,E1 -16791.06,E2 -16791.06} C_VEL
LIN {X 0,Y 292.182,Z 530.789,A -85,B 0,C 180,E1 -16793.034,E2 -16793.034} C_VEL
LIN {X 0,Y 291.139,Z 536.284,A -85,B 0,C 180,E1 -16795.16,E2 -16795.16} C_VEL
LIN {X 0,Y 290.435,Z 540.101,A -85,B 0,C 180,E1 -16797.012,E2 -16797.012} C_VEL
LIN {X 0,Y 289.756,Z 543.69,A -85,B 0,C 180,E1 -16799.379,E2 -16799.379} C_VEL
LIN {X 0,Y 289.491,Z 545.473,A -85,B 0,C 180,E1 -16800.952,E2 -16800.952} C_VEL
LIN {X 0,Y 289.223,Z 546.556,A -85,B 0,C 180,E1 -16802.504,E2 -16802.504} C_VEL
LIN {X 0,Y 289.086,Z 547.211,A -85,B 0,C 180,E1 -16804.094,E2 -16804.094} C_VEL
LIN {X 0,Y 289,Z 547.458,A -85,B 0,C 180,E1 -16805.581,E2 -16805.581} C_VEL
LIN {X 0,Y 289.037,Z 546.995,A -85,B 0,C 180,E1 -16807.515,E2 -16807.515} C_VEL
LIN {X 0,Y 289.279,Z 545.116,A -85,B 0,C 180,E1 -16810.115,E2 -16810.115} C_VEL
LIN {X 0,Y 289.675,Z 542.348,A -85,B 0,C 180,E1 -16812.346,E2 -16812.346} C_VEL
LIN {X 0,Y 290.167,Z 538.471,A -85,B 0,C 180,E1 -16814.548,E2 -16814.548} C_VEL
LIN {X 0,Y 290.865,Z 533.377,A -85,B 0,C 180,E1 -16816.73,E2 -16816.73} C_VEL
LIN {X 0,Y 291.64,Z 528.139,A -85,B 0,C 180,E1 -16818.533,E2 -16818.533} C_VEL
LIN {X 0,Y 292.686,Z 521.774,A -85,B 0,C 180,E1 -16820.324,E2 -16820.324} C_VEL
LIN {X 0,Y 293.915,Z 514.071,A -85,B 0,C 180,E1 -16822.097,E2 -16822.097} C_VEL
LIN {X 0,Y 295.192,Z 505.732,A -85,B 0,C 180,E1 -16823.678,E2 -16823.678} C_VEL
LIN {X 0,Y 296.553,Z 496.709,A -85,B 0,C 180,E1 -16825.083,E2 -16825.083} C_VEL
LIN {X 0,Y 297.802,Z 487.376,A -85,B 0,C 180,E1 -16826.279,E2 -16826.279} C_VEL
LIN {X 0,Y 298.952,Z 477.53,A -85,B 0,C 180,E1 -16827.305,E2 -16827.305} C_VEL
LIN {X 0,Y 300.047,Z 467.194,A -85,B 0,C 180,E1 -16828.155,E2 -16828.155} C_VEL
LIN {X 0,Y 300.816,Z 456.586,A -85,B 0,C 180,E1 -16828.829,E2 -16828.829} C_VEL
LIN {X 0,Y 301.531,Z 446.329,A -85,B 0,C 180,E1 -16829.291,E2 -16829.291} C_VEL
LIN {X 0,Y 302.105,Z 429.029,A -85,B 0,C 180,E1 -16829.776,E2 -16829.776} C_VEL
LIN {X 0,Y 303.593,Z 371.507,A -85,B 0,C 180,E1 -16831.162,E2 -16831.162} C_VEL
LIN {X 0,Y 300.227,Z 353.724,A -85,B 0,C 180,E1 -16831.9,E2 -16831.9} C_VEL
LIN {X 0,Y 293.937,Z 337.079,A -85,B 0,C 180,E1 -16832.913,E2 -16832.913} C_VEL
LIN {X 0,Y 293.663,Z 336.067,A -85,B 0,C 180,E1 -16833.087,E2 -16833.087} C_VEL
LIN {X 0,Y 291.775,Z 326.78,A -85,B 0,C 180,E1 -16836.483,E2 -16836.483} C_VEL
LIN {X 0,Y 291.57,Z 326.666,A -85,B 0,C 180,E1 -16839.714,E2 -16839.714} C_VEL
LIN {X 0,Y 291.524,Z 326.672,A -85,B 0,C 180,E1 -16843.95,E2 -16843.95} C_VEL
LIN {X 0,Y 291.488,Z 326.675,A -85,B 0,C 180,E1 -16846.818,E2 -16846.818} C_VEL
LIN {X 0,Y 291.453,Z 326.674,A -85,B 0,C 180,E1 -16849.875,E2 -16849.875} C_VEL
LIN {X 0,Y 291.385,Z 326.681,A -85,B 0,C 180,E1 -16854.207,E2 -16854.207} C_VEL
LIN {X 0,Y 291.423,Z 326.674,A -85,B 0,C 180,E1 -16857.272,E2 -16857.272} C_VEL
LIN {X 0,Y 291.336,Z 326.692,A -85,B 0,C 180,E1 -16860.437,E2 -16860.437} C_VEL
LIN {X 0,Y 291.346,Z 326.677,A -85,B 0,C 180,E1 -16863.698,E2 -16863.698} C_VEL
LIN {X 0,Y 291.395,Z 326.686,A -85,B 0,C 180,E1 -16867.259,E2 -16867.259} C_VEL
LIN {X 0,Y 291.336,Z 326.677,A -85,B 0,C 180,E1 -16870.642,E2 -16870.642} C_VEL
LIN {X 0,Y 291.316,Z 326.692,A -85,B 0,C 180,E1 -16874.397,E2 -16874.397} C_VEL
LIN {X 0,Y 291.327,Z 326.683,A -85,B 0,C 180,E1 -16878.404,E2 -16878.404} C_VEL
LIN {X 0,Y 291.325,Z 326.671,A -85,B 0,C 180,E1 -16881.774,E2 -16881.774} C_VEL
LIN {X 0,Y 291.371,Z 326.689,A -85,B 0,C 180,E1 -16885.095,E2 -16885.095} C_VEL
LIN {X 0,Y 291.352,Z 326.68,A -85,B 0,C 180,E1 -16887.768,E2 -16887.768} C_VEL
LIN {X 0,Y 290.754,Z 326.747,A -85,B 0,C 180,E1 -16888.921,E2 -16888.921} C_VEL
LIN {X 0,Y 287.925,Z 327.099,A -85,B 0,C 180,E1 -16890.799,E2 -16890.799} C_VEL
LIN {X 0,Y 285.469,Z 327.409,A -85,B 0,C 180,E1 -16892.323,E2 -16892.323} C_VEL
LIN {X 0,Y 284.394,Z 327.546,A -85,B 0,C 180,E1 -16893.505,E2 -16893.505} C_VEL
LIN {X 0,Y 284.297,Z 327.558,A -85,B 0,C 180,E1 -16893.906,E2 -16893.906} C_VEL
LIN {X 0,Y 284.333,Z 327.565,A -85,B 0,C 180,E1 -16896.704,E2 -16896.704} C_VEL
LIN {X 0,Y 284.378,Z 327.538,A -85,B 0,C 180,E1 -16899.904,E2 -16899.904} C_VEL
LIN {X 0,Y 284.456,Z 327.533,A -85,B 0,C 180,E1 -16904.487,E2 -16904.487} C_VEL
LIN {X 0,Y 284.485,Z 327.544,A -85,B 0,C 180,E1 -16908.601,E2 -16908.601} C_VEL
LIN {X 0,Y 284.61,Z 327.508,A -85,B 0,C 180,E1 -16911.479,E2 -16911.479} C_VEL
LIN {X 0,Y 284.571,Z 327.5,A -85,B 0,C 180,E1 -16914.33,E2 -16914.33} C_VEL
LIN {X 0,Y 284.84,Z 327.503,A -85,B 0,C 180,E1 -16918.586,E2 -16918.586} C_VEL
LIN {X 0,Y 284.847,Z 327.493,A -85,B 0,C 180,E1 -16921.413,E2 -16921.413} C_VEL
LIN {X 0,Y 284.66,Z 327.507,A -85,B 0,C 180,E1 -16927.091,E2 -16927.091} C_VEL
LIN {X 0,Y 284.515,Z 327.543,A -85,B 0,C 180,E1 -16929.957,E2 -16929.957} C_VEL
LIN {X 0,Y 284.419,Z 327.529,A -85,B 0,C 180,E1 -16934.306,E2 -16934.306} C_VEL
LIN {X 0,Y 284.324,Z 327.566,A -85,B 0,C 180,E1 -16938.743,E2 -16938.743} C_VEL
LIN {X 0,Y 284.327,Z 327.546,A -85,B 0,C 180,E1 -16943.296,E2 -16943.296} C_VEL
LIN {X 0,Y 284.329,Z 327.568,A -85,B 0,C 180,E1 -16947.146,E2 -16947.146} C_VEL
LIN {X 0,Y 284.296,Z 327.562,A -85,B 0,C 180,E1 -16950.091,E2 -16950.091} C_VEL
LIN {X 0,Y 284.304,Z 327.563,A -85,B 0,C 180,E1 -16952.945,E2 -16952.945} C_VEL
LIN {X 0,Y 284.318,Z 327.56,A -85,B 0,C 180,E1 -16956.388,E2 -16956.388} C_VEL
LIN {X 0,Y 284.253,Z 327.579,A -85,B 0,C 180,E1 -16960.003,E2 -16960.003} C_VEL
LIN {X 0,Y 284.232,Z 327.579,A -85,B 0,C 180,E1 -16964.187,E2 -16964.187} C_VEL
LIN {X 0,Y 284.238,Z 327.58,A -85,B 0,C 180,E1 -16968.118,E2 -16968.118} C_VEL
LIN {X 0,Y 284.307,Z 327.569,A -85,B 0,C 180,E1 -16972.281,E2 -16972.281} C_VEL
LIN {X 0,Y 284.307,Z 327.561,A -85,B 0,C 180,E1 -16976.207,E2 -16976.207} C_VEL
LIN {X 0,Y 284.347,Z 327.805,A -85,B 0,C 180,E1 -16976.902,E2 -16976.902} C_VEL
LIN {X 0,Y 286.546,Z 338.092,A -85,B 0,C 180,E1 -16980.624,E2 -16980.624} C_VEL
LIN {X 0,Y 287.71,Z 343.725,A -85,B 0,C 180,E1 -16982.511,E2 -16982.511} C_VEL
LIN {X 0,Y 290.803,Z 352.099,A -85,B 0,C 180,E1 -16983.074,E2 -16983.074} C_VEL
LIN {X 0,Y 292.232,Z 356.641,A -85,B 0,C 180,E1 -16983.326,E2 -16983.326} C_VEL
LIN {X 0,Y 296.774,Z 384.923,A -85,B 0,C 180,E1 -16984.479,E2 -16984.479} C_VEL
LIN {X 0,Y 294.934,Z 449.761,A -85,B 0,C 180,E1 -16986.103,E2 -16986.103} C_VEL
LIN {X 0,Y 294.448,Z 459.576,A -85,B 0,C 180,E1 -16986.481,E2 -16986.481} C_VEL
LIN {X 0,Y 293.655,Z 469.545,A -85,B 0,C 180,E1 -16987.02,E2 -16987.02} C_VEL
LIN {X 0,Y 292.589,Z 479.897,A -85,B 0,C 180,E1 -16987.77,E2 -16987.77} C_VEL
LIN {X 0,Y 291.332,Z 490.606,A -85,B 0,C 180,E1 -16988.786,E2 -16988.786} C_VEL
LIN {X 0,Y 289.965,Z 500.626,A -85,B 0,C 180,E1 -16989.979,E2 -16989.979} C_VEL
LIN {X 0,Y 288.732,Z 508.979,A -85,B 0,C 180,E1 -16991.185,E2 -16991.185} C_VEL
LIN {X 0,Y 287.515,Z 517.112,A -85,B 0,C 180,E1 -16992.596,E2 -16992.596} C_VEL
LIN {X 0,Y 286.153,Z 525.325,A -85,B 0,C 180,E1 -16994.326,E2 -16994.326} C_VEL
LIN {X 0,Y 285.018,Z 532.24,A -85,B 0,C 180,E1 -16996.089,E2 -16996.089} C_VEL
LIN {X 0,Y 284.065,Z 538.015,A -85,B 0,C 180,E1 -16997.86,E2 -16997.86} C_VEL
LIN {X 0,Y 283.257,Z 543.604,A -85,B 0,C 180,E1 -16999.998,E2 -16999.998} C_VEL
LIN {X 0,Y 282.729,Z 547.993,A -85,B 0,C 180,E1 -17002.142,E2 -17002.142} C_VEL
LIN {X 0,Y 282.392,Z 551.606,A -85,B 0,C 180,E1 -17004.554,E2 -17004.554} C_VEL
LIN {X 0,Y 282.305,Z 552.931,A -85,B 0,C 180,E1 -17005.717,E2 -17005.717} C_VEL
LIN {X 0,Y 282.292,Z 554.998,A -85,B 0,C 180,E1 -17008.573,E2 -17008.573} C_VEL
LIN {X 0,Y 282.293,Z 555.312,A -85,B 0,C 180,E1 -17011.426,E2 -17011.426} C_VEL
LIN {X 0,Y 282.302,Z 554.976,A -85,B 0,C 180,E1 -17012.854,E2 -17012.854} C_VEL
LIN {X 0,Y 282.439,Z 552.908,A -85,B 0,C 180,E1 -17015.712,E2 -17015.712} C_VEL
LIN {X 0,Y 282.764,Z 550.305,A -85,B 0,C 180,E1 -17017.857,E2 -17017.857} C_VEL
LIN {X 0,Y 283.356,Z 546.692,A -85,B 0,C 180,E1 -17019.998,E2 -17019.998} C_VEL
LIN {X 0,Y 284.253,Z 541.967,A -85,B 0,C 180,E1 -17022.131,E2 -17022.131} C_VEL
LIN {X 0,Y 285.471,Z 535.985,A -85,B 0,C 180,E1 -17024.252,E2 -17024.252} C_VEL
LIN {X 0,Y 286.817,Z 529.943,A -85,B 0,C 180,E1 -17026.001,E2 -17026.001} C_VEL
LIN {X 0,Y 288.373,Z 521.792,A -85,B 0,C 180,E1 -17027.926,E2 -17027.926} C_VEL
LIN {X 0,Y 289.936,Z 513.839,A -85,B 0,C 180,E1 -17029.469,E2 -17029.469} C_VEL
LIN {X 0,Y 291.54,Z 505.381,A -85,B 0,C 180,E1 -17030.828,E2 -17030.828} C_VEL
LIN {X 0,Y 293.371,Z 495.057,A -85,B 0,C 180,E1 -17032.167,E2 -17032.167} C_VEL
LIN {X 0,Y 294.837,Z 485.607,A -85,B 0,C 180,E1 -17033.16,E2 -17033.16} C_VEL
LIN {X 0,Y 296.213,Z 474.693,A -85,B 0,C 180,E1 -17034.066,E2 -17034.066} C_VEL
LIN {X 0,Y 297.279,Z 464.385,A -85,B 0,C 180,E1 -17034.718,E2 -17034.718} C_VEL
LIN {X 0,Y 298.247,Z 453.417,A -85,B 0,C 180,E1 -17035.2,E2 -17035.2} C_VEL
LIN {X 0,Y 298.854,Z 434.982,A -85,B 0,C 180,E1 -17035.73,E2 -17035.73} C_VEL
LIN {X 0,Y 300.368,Z 385.701,A -85,B 0,C 180,E1 -17036.955,E2 -17036.955} C_VEL
LIN {X 0,Y 296.765,Z 363.814,A -85,B 0,C 180,E1 -17037.99,E2 -17037.99} C_VEL
LIN {X 0,Y 295.298,Z 359.495,A -85,B 0,C 180,E1 -17038.287,E2 -17038.287} C_VEL
LIN {X 0,Y 289.265,Z 345.896,A -85,B 0,C 180,E1 -17039.44,E2 -17039.44} C_VEL
LIN {X 0,Y 288.012,Z 342.817,A -85,B 0,C 180,E1 -17039.776,E2 -17039.776} C_VEL
LIN {X 0,Y 285.796,Z 333.205,A -85,B 0,C 180,E1 -17043.271,E2 -17043.271} C_VEL
LIN {X 0,Y 284.33,Z 327.609,A -85,B 0,C 180,E1 -17045.586,E2 -17045.586} C_VEL
LIN {X 0,Y 284.31,Z 327.571,A -85,B 0,C 180,E1 -17048.169,E2 -17048.169} C_VEL
LIN {X 0,Y 284.267,Z 327.576,A -85,B 0,C 180,E1 -17052.125,E2 -17052.125} C_VEL
LIN {X 0,Y 284.253,Z 327.574,A -85,B 0,C 180,E1 -17056.189,E2 -17056.189} C_VEL
LIN {X 0,Y 284.305,Z 327.572,A -85,B 0,C 180,E1 -17060.024,E2 -17060.024} C_VEL
LIN {X 0,Y 284.329,Z 327.568,A -85,B 0,C 180,E1 -17063.614,E2 -17063.614} C_VEL
LIN {X 0,Y 284.307,Z 327.569,A -85,B 0,C 180,E1 -17067.19,E2 -17067.19} C_VEL
LIN {X 0,Y 284.355,Z 327.565,A -85,B 0,C 180,E1 -17070.376,E2 -17070.376} C_VEL
LIN {X 0,Y 284.377,Z 327.557,A -85,B 0,C 180,E1 -17073.587,E2 -17073.587} C_VEL
LIN {X 0,Y 284.366,Z 327.553,A -85,B 0,C 180,E1 -17076.707,E2 -17076.707} C_VEL
LIN {X 0,Y 284.403,Z 327.548,A -85,B 0,C 180,E1 -17081.262,E2 -17081.262} C_VEL
LIN {X 0,Y 284.493,Z 327.545,A -85,B 0,C 180,E1 -17084.459,E2 -17084.459} C_VEL
LIN {X 0,Y 284.489,Z 327.546,A -85,B 0,C 180,E1 -17088.602,E2 -17088.602} C_VEL
LIN {X 0,Y 284.661,Z 327.513,A -85,B 0,C 180,E1 -17091.482,E2 -17091.482} C_VEL
LIN {X 0,Y 284.603,Z 327.53,A -85,B 0,C 180,E1 -17094.332,E2 -17094.332} C_VEL
LIN {X 0,Y 284.857,Z 327.501,A -85,B 0,C 180,E1 -17098.587,E2 -17098.587} C_VEL
LIN {X 0,Y 284.857,Z 327.496,A -85,B 0,C 180,E1 -17101.414,E2 -17101.414} C_VEL
LIN {X 0,Y 284.7,Z 327.523,A -85,B 0,C 180,E1 -17107.09,E2 -17107.09} C_VEL
LIN {X 0,Y 284.568,Z 327.536,A -85,B 0,C 180,E1 -17109.956,E2 -17109.956} C_VEL
LIN {X 0,Y 284.483,Z 327.549,A -85,B 0,C 180,E1 -17114.303,E2 -17114.303} C_VEL
LIN {X 0,Y 284.424,Z 327.554,A -85,B 0,C 180,E1 -17117.249,E2 -17117.249} C_VEL
LIN {X 0,Y 284.378,Z 327.562,A -85,B 0,C 180,E1 -17120.243,E2 -17120.243} C_VEL
LIN {X 0,Y 284.323,Z 327.567,A -85,B 0,C 180,E1 -17124.848,E2 -17124.848} C_VEL
LIN {X 0,Y 284.315,Z 327.555,A -85,B 0,C 180,E1 -17128.013,E2 -17128.013} C_VEL
LIN {X 0,Y 284.294,Z 327.562,A -85,B 0,C 180,E1 -17131.275,E2 -17131.275} C_VEL
LIN {X 0,Y 284.356,Z 327.678,A -85,B 0,C 180,E1 -17132.825,E2 -17132.825} C_VEL
LIN {X 0,Y 286.385,Z 335.593,A -85,B 0,C 180,E1 -17135.92,E2 -17135.92} C_VEL
LIN {X 0,Y 286.825,Z 336.913,A -85,B 0,C 180,E1 -17136.2,E2 -17136.2} C_VEL
LIN {X 0,Y 293.981,Z 351.777,A -85,B 0,C 180,E1 -17137.574,E2 -17137.574} C_VEL
LIN {X 0,Y 299.061,Z 364.25,A -85,B 0,C 180,E1 -17138.531,E2 -17138.531} C_VEL
LIN {X 0,Y 300.75,Z 373.968,A -85,B 0,C 180,E1 -17138.999,E2 -17138.999} C_VEL
LIN {X 0,Y 298.433,Z 442.455,A -85,B 0,C 180,E1 -17140.722,E2 -17140.722} C_VEL
LIN {X 0,Y 297.778,Z 452.512,A -85,B 0,C 180,E1 -17141.108,E2 -17141.108} C_VEL
LIN {X 0,Y 297.03,Z 461.769,A -85,B 0,C 180,E1 -17141.61,E2 -17141.61} C_VEL
LIN {X 0,Y 295.935,Z 472.225,A -85,B 0,C 180,E1 -17142.369,E2 -17142.369} C_VEL
LIN {X 0,Y 294.567,Z 482.349,A -85,B 0,C 180,E1 -17143.308,E2 -17143.308} C_VEL
LIN {X 0,Y 293.016,Z 492.335,A -85,B 0,C 180,E1 -17144.475,E2 -17144.475} C_VEL
LIN {X 0,Y 291.27,Z 502.15,A -85,B 0,C 180,E1 -17145.9,E2 -17145.9} C_VEL
LIN {X 0,Y 289.751,Z 509.762,A -85,B 0,C 180,E1 -17147.223,E2 -17147.223} C_VEL
LIN {X 0,Y 288.185,Z 517.371,A -85,B 0,C 180,E1 -17148.818,E2 -17148.818} C_VEL
LIN {X 0,Y 286.585,Z 525.137,A -85,B 0,C 180,E1 -17150.832,E2 -17150.832} C_VEL
LIN {X 0,Y 285.459,Z 530.373,A -85,B 0,C 180,E1 -17152.458,E2 -17152.458} C_VEL
LIN {X 0,Y 284.277,Z 536.052,A -85,B 0,C 180,E1 -17154.671,E2 -17154.671} C_VEL
LIN {X 0,Y 283.356,Z 540.532,A -85,B 0,C 180,E1 -17156.93,E2 -17156.93} C_VEL
LIN {X 0,Y 282.853,Z 543.094,A -85,B 0,C 180,E1 -17158.548,E2 -17158.548} C_VEL
LIN {X 0,Y 282.444,Z 545.377,A -85,B 0,C 180,E1 -17160.564,E2 -17160.564} C_VEL
LIN {X 0,Y 282.02,Z 547.267,A -85,B 0,C 180,E1 -17163.784,E2 -17163.784} C_VEL
LIN {X 0,Y 281.94,Z 547.516,A -85,B 0,C 180,E1 -17164.928,E2 -17164.928} C_VEL
LIN {X 0,Y 281.964,Z 546.781,A -85,B 0,C 180,E1 -17168.045,E2 -17168.045} C_VEL
LIN {X 0,Y 282.1,Z 545.727,A -85,B 0,C 180,E1 -17169.587,E2 -17169.587} C_VEL
LIN {X 0,Y 282.363,Z 544.113,A -85,B 0,C 180,E1 -17171.121,E2 -17171.121} C_VEL
LIN {X 0,Y 282.794,Z 540.902,A -85,B 0,C 180,E1 -17173.394,E2 -17173.394} C_VEL
LIN {X 0,Y 283.3,Z 537.173,A -85,B 0,C 180,E1 -17175.352,E2 -17175.352} C_VEL
LIN {X 0,Y 283.928,Z 532.955,A -85,B 0,C 180,E1 -17177.128,E2 -17177.128} C_VEL
LIN {X 0,Y 284.766,Z 527.599,A -85,B 0,C 180,E1 -17178.973,E2 -17178.973} C_VEL
LIN {X 0,Y 285.843,Z 521.112,A -85,B 0,C 180,E1 -17180.804,E2 -17180.804} C_VEL
LIN {X 0,Y 286.909,Z 515.013,A -85,B 0,C 180,E1 -17182.257,E2 -17182.257} C_VEL
LIN {X 0,Y 288.351,Z 505.79,A -85,B 0,C 180,E1 -17184.054,E2 -17184.054} C_VEL
LIN {X 0,Y 289.67,Z 497.435,A -85,B 0,C 180,E1 -17185.396,E2 -17185.396} C_VEL
LIN {X 0,Y 291.051,Z 487.417,A -85,B 0,C 180,E1 -17186.712,E2 -17186.712} C_VEL
LIN {X 0,Y 292.252,Z 477.548,A -85,B 0,C 180,E1 -17187.761,E2 -17187.761} C_VEL
LIN {X 0,Y 293.384,Z 467.189,A -85,B 0,C 180,E1 -17188.627,E2 -17188.627} C_VEL
LIN {X 0,Y 294.184,Z 456.546,A -85,B 0,C 180,E1 -17189.316,E2 -17189.316} C_VEL
LIN {X 0,Y 294.925,Z 446.222,A -85,B 0,C 180,E1 -17189.787,E2 -17189.787} C_VEL
LIN {X 0,Y 295.517,Z 429.338,A -85,B 0,C 180,E1 -17190.269,E2 -17190.269} C_VEL
LIN {X 0,Y 296.99,Z 372.004,A -85,B 0,C 180,E1 -17191.682,E2 -17191.682} C_VEL
LIN {X 0,Y 293.932,Z 355.981,A -85,B 0,C 180,E1 -17192.37,E2 -17192.37} C_VEL
LIN {X 0,Y 287.253,Z 338.706,A -85,B 0,C 180,E1 -17193.442,E2 -17193.442} C_VEL
LIN {X 0,Y 286.455,Z 336.454,A -85,B 0,C 180,E1 -17193.666,E2 -17193.666} C_VEL
LIN {X 0,Y 284.68,Z 327.591,A -85,B 0,C 180,E1 -17197.002,E2 -17197.002} C_VEL
LIN {X 0,Y 284.516,Z 327.546,A -85,B 0,C 180,E1 -17199.957,E2 -17199.957} C_VEL
LIN {X 0,Y 284.484,Z 327.547,A -85,B 0,C 180,E1 -17204.303,E2 -17204.303} C_VEL
LIN {X 0,Y 284.425,Z 327.555,A -85,B 0,C 180,E1 -17207.249,E2 -17207.249} C_VEL
LIN {X 0,Y 284.379,Z 327.558,A -85,B 0,C 180,E1 -17210.242,E2 -17210.242} C_VEL
LIN {X 0,Y 284.34,Z 327.565,A -85,B 0,C 180,E1 -17214.847,E2 -17214.847} C_VEL
LIN {X 0,Y 284.33,Z 327.554,A -85,B 0,C 180,E1 -17218.011,E2 -17218.011} C_VEL
LIN {X 0,Y 284.296,Z 327.574,A -85,B 0,C 180,E1 -17221.275,E2 -17221.275} C_VEL
LIN {X 0,Y 284.363,Z 327.548,A -85,B 0,C 180,E1 -17225.354,E2 -17225.354} C_VEL
LIN {X 0,Y 284.325,Z 327.568,A -85,B 0,C 180,E1 -17228.167,E2 -17228.167} C_VEL
LIN {X 0,Y 284.271,Z 327.553,A -85,B 0,C 180,E1 -17232.124,E2 -17232.124} C_VEL
LIN {X 0,Y 284.271,Z 327.575,A -85,B 0,C 180,E1 -17236.192,E2 -17236.192} C_VEL
LIN {X 0,Y 284.308,Z 327.542,A -85,B 0,C 180,E1 -17240.024,E2 -17240.024} C_VEL
LIN {X 0,Y 284.33,Z 327.563,A -85,B 0,C 180,E1 -17243.613,E2 -17243.613} C_VEL
LIN {X 0,Y 284.276,Z 327.56,A -85,B 0,C 180,E1 -17247.759,E2 -17247.759} C_VEL
LIN {X 0,Y 284.339,Z 327.528,A -85,B 0,C 180,E1 -17250.373,E2 -17250.373} C_VEL
LIN {X 0,Y 284.297,Z 327.558,A -85,B 0,C 180,E1 -17253.906,E2 -17253.906} C_VEL
LIN {X 0,Y 283.611,Z 327.654,A -85,B 0,C 180,E1 -17255.088,E2 -17255.088} C_VEL
LIN {X 0,Y 280.779,Z 328.006,A -85,B 0,C 180,E1 -17257.015,E2 -17257.015} C_VEL
LIN {X 0,Y 278.396,Z 328.297,A -85,B 0,C 180,E1 -17258.58,E2 -17258.58} C_VEL
LIN {X 0,Y 277.383,Z 328.411,A -85,B 0,C 180,E1 -17259.792,E2 -17259.792} C_VEL
LIN {X 0,Y 277.304,Z 328.413,A -85,B 0,C 180,E1 -17260.202,E2 -17260.202} C_VEL
LIN {X 0,Y 277.396,Z 328.411,A -85,B 0,C 180,E1 -17264.314,E2 -17264.314} C_VEL
LIN {X 0,Y 277.432,Z 328.423,A -85,B 0,C 180,E1 -17268.307,E2 -17268.307} C_VEL
LIN {X 0,Y 277.572,Z 328.387,A -85,B 0,C 180,E1 -17271.262,E2 -17271.262} C_VEL
LIN {X 0,Y 277.541,Z 328.373,A -85,B 0,C 180,E1 -17274.186,E2 -17274.186} C_VEL
LIN {X 0,Y 277.807,Z 328.379,A -85,B 0,C 180,E1 -17278.55,E2 -17278.55} C_VEL
LIN {X 0,Y 277.813,Z 328.369,A -85,B 0,C 180,E1 -17281.449,E2 -17281.449} C_VEL
LIN {X 0,Y 277.617,Z 328.386,A -85,B 0,C 180,E1 -17287.271,E2 -17287.271} C_VEL
LIN {X 0,Y 277.456,Z 328.422,A -85,B 0,C 180,E1 -17290.213,E2 -17290.213} C_VEL
LIN {X 0,Y 277.372,Z 328.404,A -85,B 0,C 180,E1 -17294.677,E2 -17294.677} C_VEL
LIN {X 0,Y 277.28,Z 328.444,A -85,B 0,C 180,E1 -17299.238,E2 -17299.238} C_VEL
LIN {X 0,Y 277.282,Z 328.421,A -85,B 0,C 180,E1 -17303.924,E2 -17303.924} C_VEL
LIN {X 0,Y 277.269,Z 328.446,A -85,B 0,C 180,E1 -17307.482,E2 -17307.482} C_VEL
LIN {X 0,Y 277.248,Z 328.435,A -85,B 0,C 180,E1 -17310.472,E2 -17310.472} C_VEL
LIN {X 0,Y 277.245,Z 328.451,A -85,B 0,C 180,E1 -17313.895,E2 -17313.895} C_VEL
LIN {X 0,Y 277.231,Z 328.439,A -85,B 0,C 180,E1 -17317.474,E2 -17317.474} C_VEL
LIN {X 0,Y 277.175,Z 328.456,A -85,B 0,C 180,E1 -17321.242,E2 -17321.242} C_VEL
LIN {X 0,Y 277.172,Z 328.457,A -85,B 0,C 180,E1 -17325.232,E2 -17325.232} C_VEL
LIN {X 0,Y 277.182,Z 328.456,A -85,B 0,C 180,E1 -17328.758,E2 -17328.758} C_VEL
LIN {X 0,Y 277.253,Z 328.449,A -85,B 0,C 180,E1 -17332.528,E2 -17332.528} C_VEL
LIN {X 0,Y 277.273,Z 328.528,A -85,B 0,C 180,E1 -17336.304,E2 -17336.304} C_VEL
LIN {X 0,Y 279.295,Z 337.69,A -85,B 0,C 180,E1 -17339.783,E2 -17339.783} C_VEL
LIN {X 0,Y 280.441,Z 343.625,A -85,B 0,C 180,E1 -17341.823,E2 -17341.823} C_VEL
LIN {X 0,Y 282.283,Z 348.632,A -85,B 0,C 180,E1 -17342.211,E2 -17342.211} C_VEL
LIN {X 0,Y 285.845,Z 358.273,A -85,B 0,C 180,E1 -17342.806,E2 -17342.806} C_VEL
LIN {X 0,Y 290.211,Z 385.272,A -85,B 0,C 180,E1 -17343.943,E2 -17343.943} C_VEL
LIN {X 0,Y 288.308,Z 450.246,A -85,B 0,C 180,E1 -17345.614,E2 -17345.614} C_VEL
LIN {X 0,Y 287.779,Z 459.85,A -85,B 0,C 180,E1 -17345.998,E2 -17345.998} C_VEL
LIN {X 0,Y 286.991,Z 469.724,A -85,B 0,C 180,E1 -17346.55,E2 -17346.55} C_VEL
LIN {X 0,Y 285.777,Z 480.952,A -85,B 0,C 180,E1 -17347.402,E2 -17347.402} C_VEL
LIN {X 0,Y 284.693,Z 489.93,A -85,B 0,C 180,E1 -17348.266,E2 -17348.266} C_VEL
LIN {X 0,Y 283.239,Z 500.055,A -85,B 0,C 180,E1 -17349.483,E2 -17349.483} C_VEL
LIN {X 0,Y 281.805,Z 509.522,A -85,B 0,C 180,E1 -17350.893,E2 -17350.893} C_VEL
LIN {X 0,Y 280.436,Z 518.319,A -85,B 0,C 180,E1 -17352.498,E2 -17352.498} C_VEL
LIN {X 0,Y 279.279,Z 524.964,A -85,B 0,C 180,E1 -17353.93,E2 -17353.93} C_VEL
LIN {X 0,Y 278.079,Z 531.926,A -85,B 0,C 180,E1 -17355.734,E2 -17355.734} C_VEL
LIN {X 0,Y 277.067,Z 537.743,A -85,B 0,C 180,E1 -17357.549,E2 -17357.549} C_VEL
LIN {X 0,Y 276.241,Z 543.371,A -85,B 0,C 180,E1 -17359.741,E2 -17359.741} C_VEL
LIN {X 0,Y 275.676,Z 547.793,A -85,B 0,C 180,E1 -17361.94,E2 -17361.94} C_VEL
LIN {X 0,Y 275.3,Z 551.672,A -85,B 0,C 180,E1 -17364.626,E2 -17364.626} C_VEL
LIN {X 0,Y 275.21,Z 553.961,A -85,B 0,C 180,E1 -17367.072,E2 -17367.072} C_VEL
LIN {X 0,Y 275.219,Z 554.878,A -85,B 0,C 180,E1 -17368.537,E2 -17368.537} C_VEL
LIN {X 0,Y 275.219,Z 555.226,A -85,B 0,C 180,E1 -17371.463,E2 -17371.463} C_VEL
LIN {X 0,Y 275.215,Z 554.892,A -85,B 0,C 180,E1 -17372.927,E2 -17372.927} C_VEL
LIN {X 0,Y 275.377,Z 552.882,A -85,B 0,C 180,E1 -17375.859,E2 -17375.859} C_VEL
LIN {X 0,Y 275.726,Z 550.314,A -85,B 0,C 180,E1 -17378.059,E2 -17378.059} C_VEL
LIN {X 0,Y 276.359,Z 546.734,A -85,B 0,C 180,E1 -17380.254,E2 -17380.254} C_VEL
LIN {X 0,Y 277.302,Z 542.046,A -85,B 0,C 180,E1 -17382.44,E2 -17382.44} C_VEL
LIN {X 0,Y 278.606,Z 536.103,A -85,B 0,C 180,E1 -17384.611,E2 -17384.611} C_VEL
LIN {X 0,Y 280.304,Z 528.685,A -85,B 0,C 180,E1 -17386.758,E2 -17386.758} C_VEL
LIN {X 0,Y 281.502,Z 522.599,A -85,B 0,C 180,E1 -17388.247,E2 -17388.247} C_VEL
LIN {X 0,Y 283.27,Z 514.112,A -85,B 0,C 180,E1 -17389.946,E2 -17389.946} C_VEL
LIN {X 0,Y 285.16,Z 504.508,A -85,B 0,C 180,E1 -17391.506,E2 -17391.506} C_VEL
LIN {X 0,Y 286.848,Z 495.524,A -85,B 0,C 180,E1 -17392.699,E2 -17392.699} C_VEL
LIN {X 0,Y 288.367,Z 486.232,A -85,B 0,C 180,E1 -17393.711,E2 -17393.711} C_VEL
LIN {X 0,Y 289.788,Z 475.553,A -85,B 0,C 180,E1 -17394.635,E2 -17394.635} C_VEL
LIN {X 0,Y 291.044,Z 463.991,A -85,B 0,C 180,E1 -17395.38,E2 -17395.38} C_VEL
LIN {X 0,Y 291.993,Z 453.408,A -85,B 0,C 180,E1 -17395.856,E2 -17395.856} C_VEL
LIN {X 0,Y 292.658,Z 434.381,A -85,B 0,C 180,E1 -17396.413,E2 -17396.413} C_VEL
LIN {X 0,Y 294.222,Z 386.739,A -85,B 0,C 180,E1 -17397.618,E2 -17397.618} C_VEL
LIN {X 0,Y 290.701,Z 365.269,A -85,B 0,C 180,E1 -17398.669,E2 -17398.669} C_VEL
LIN {X 0,Y 284.217,Z 350.131,A -85,B 0,C 180,E1 -17399.968,E2 -17399.968} C_VEL
LIN {X 0,Y 280.83,Z 342.818,A -85,B 0,C 180,E1 -17400.705,E2 -17400.705} C_VEL
LIN {X 0,Y 278.64,Z 333.771,A -85,B 0,C 180,E1 -17404.138,E2 -17404.138} C_VEL
LIN {X 0,Y 277.315,Z 328.509,A -85,B 0,C 180,E1 -17406.393,E2 -17406.393} C_VEL
LIN {X 0,Y 277.22,Z 328.439,A -85,B 0,C 180,E1 -17410.488,E2 -17410.488} C_VEL
LIN {X 0,Y 277.199,Z 328.458,A -85,B 0,C 180,E1 -17414.774,E2 -17414.774} C_VEL
LIN {X 0,Y 277.208,Z 328.449,A -85,B 0,C 180,E1 -17418.764,E2 -17418.764} C_VEL
LIN {X 0,Y 277.264,Z 328.447,A -85,B 0,C 180,E1 -17422.531,E2 -17422.531} C_VEL
LIN {X 0,Y 277.246,Z 328.448,A -85,B 0,C 180,E1 -17426.105,E2 -17426.105} C_VEL
LIN {X 0,Y 277.261,Z 328.444,A -85,B 0,C 180,E1 -17429.539,E2 -17429.539} C_VEL
LIN {X 0,Y 277.357,Z 328.427,A -85,B 0,C 180,E1 -17432.864,E2 -17432.864} C_VEL
LIN {X 0,Y 277.329,Z 328.434,A -85,B 0,C 180,E1 -17436.08,E2 -17436.08} C_VEL
LIN {X 0,Y 277.345,Z 328.429,A -85,B 0,C 180,E1 -17440.767,E2 -17440.767} C_VEL
LIN {X 0,Y 277.435,Z 328.418,A -85,B 0,C 180,E1 -17445.326,E2 -17445.326} C_VEL
LIN {X 0,Y 277.507,Z 328.411,A -85,B 0,C 180,E1 -17449.789,E2 -17449.789} C_VEL
LIN {X 0,Y 277.655,Z 328.398,A -85,B 0,C 180,E1 -17452.73,E2 -17452.73} C_VEL
LIN {X 0,Y 277.823,Z 328.378,A -85,B 0,C 180,E1 -17458.551,E2 -17458.551} C_VEL
LIN {X 0,Y 277.823,Z 328.373,A -85,B 0,C 180,E1 -17461.45,E2 -17461.45} C_VEL
LIN {X 0,Y 277.655,Z 328.399,A -85,B 0,C 180,E1 -17467.271,E2 -17467.271} C_VEL
LIN {X 0,Y 277.508,Z 328.416,A -85,B 0,C 180,E1 -17470.212,E2 -17470.212} C_VEL
LIN {X 0,Y 277.436,Z 328.426,A -85,B 0,C 180,E1 -17474.674,E2 -17474.674} C_VEL
LIN {X 0,Y 277.343,Z 328.432,A -85,B 0,C 180,E1 -17479.234,E2 -17479.234} C_VEL
LIN {X 0,Y 277.285,Z 328.443,A -85,B 0,C 180,E1 -17484.155,E2 -17484.155} C_VEL
LIN {X 0,Y 277.309,Z 328.427,A -85,B 0,C 180,E1 -17487.499,E2 -17487.499} C_VEL
LIN {X 0,Y 277.295,Z 328.48,A -85,B 0,C 180,E1 -17491.922,E2 -17491.922} C_VEL
LIN {X 0,Y 278.291,Z 332.198,A -85,B 0,C 180,E1 -17493.552,E2 -17493.552} C_VEL
LIN {X 0,Y 279.389,Z 336.419,A -85,B 0,C 180,E1 -17495.129,E2 -17495.129} C_VEL
LIN {X 0,Y 286.622,Z 351.061,A -85,B 0,C 180,E1 -17496.627,E2 -17496.627} C_VEL
LIN {X 0,Y 293.17,Z 366.636,A -85,B 0,C 180,E1 -17497.914,E2 -17497.914} C_VEL
LIN {X 0,Y 294.636,Z 375.914,A -85,B 0,C 180,E1 -17498.358,E2 -17498.358} C_VEL
LIN {X 0,Y 292.173,Z 443.028,A -85,B 0,C 180,E1 -17500.076,E2 -17500.076} C_VEL
LIN {X 0,Y 291.522,Z 452.761,A -85,B 0,C 180,E1 -17500.463,E2 -17500.463} C_VEL
LIN {X 0,Y 290.707,Z 462.145,A -85,B 0,C 180,E1 -17500.985,E2 -17500.985} C_VEL
LIN {X 0,Y 289.449,Z 473.333,A -85,B 0,C 180,E1 -17501.831,E2 -17501.831} C_VEL
LIN {X 0,Y 288.152,Z 482.588,A -85,B 0,C 180,E1 -17502.714,E2 -17502.714} C_VEL
LIN {X 0,Y 286.541,Z 492.548,A -85,B 0,C 180,E1 -17503.907,E2 -17503.907} C_VEL
LIN {X 0,Y 284.881,Z 501.576,A -85,B 0,C 180,E1 -17505.232,E2 -17505.232} C_VEL
LIN {X 0,Y 283.367,Z 508.937,A -85,B 0,C 180,E1 -17506.509,E2 -17506.509} C_VEL
LIN {X 0,Y 281.623,Z 516.996,A -85,B 0,C 180,E1 -17508.208,E2 -17508.208} C_VEL
LIN {X 0,Y 279.93,Z 524.617,A -85,B 0,C 180,E1 -17510.193,E2 -17510.193} C_VEL
LIN {X 0,Y 278.63,Z 530.346,A -85,B 0,C 180,E1 -17511.998,E2 -17511.998} C_VEL
LIN {X 0,Y 277.307,Z 536.224,A -85,B 0,C 180,E1 -17514.345,E2 -17514.345} C_VEL
LIN {X 0,Y 276.561,Z 539.643,A -85,B 0,C 180,E1 -17516.009,E2 -17516.009} C_VEL
LIN {X 0,Y 275.776,Z 543.452,A -85,B 0,C 180,E1 -17518.505,E2 -17518.505} C_VEL
LIN {X 0,Y 275.27,Z 545.97,A -85,B 0,C 180,E1 -17520.981,E2 -17520.981} C_VEL
LIN {X 0,Y 274.934,Z 547.328,A -85,B 0,C 180,E1 -17523.469,E2 -17523.469} C_VEL
LIN {X 0,Y 274.826,Z 547.565,A -85,B 0,C 180,E1 -17525.848,E2 -17525.848} C_VEL
LIN {X 0,Y 274.86,Z 547.2,A -85,B 0,C 180,E1 -17527.447,E2 -17527.447} C_VEL
LIN {X 0,Y 275.17,Z 544.859,A -85,B 0,C 180,E1 -17530.608,E2 -17530.608} C_VEL
LIN {X 0,Y 275.439,Z 543.099,A -85,B 0,C 180,E1 -17532.171,E2 -17532.171} C_VEL
LIN {X 0,Y 275.994,Z 539.269,A -85,B 0,C 180,E1 -17534.568,E2 -17534.568} C_VEL
LIN {X 0,Y 276.828,Z 533.53,A -85,B 0,C 180,E1 -17537.165,E2 -17537.165} C_VEL
LIN {X 0,Y 277.694,Z 528.274,A -85,B 0,C 180,E1 -17539.058,E2 -17539.058} C_VEL
LIN {X 0,Y 278.832,Z 521.725,A -85,B 0,C 180,E1 -17540.98,E2 -17540.98} C_VEL
LIN {X 0,Y 280.169,Z 514.164,A -85,B 0,C 180,E1 -17542.795,E2 -17542.795} C_VEL
LIN {X 0,Y 281.362,Z 506.868,A -85,B 0,C 180,E1 -17544.266,E2 -17544.266} C_VEL
LIN {X 0,Y 282.785,Z 498.12,A -85,B 0,C 180,E1 -17545.724,E2 -17545.724} C_VEL
LIN {X 0,Y 284.144,Z 488.926,A -85,B 0,C 180,E1 -17546.987,E2 -17546.987} C_VEL
LIN {X 0,Y 285.373,Z 479.396,A -85,B 0,C 180,E1 -17548.06,E2 -17548.06} C_VEL
LIN {X 0,Y 286.63,Z 468.313,A -85,B 0,C 180,E1 -17549.034,E2 -17549.034} C_VEL
LIN {X 0,Y 287.579,Z 456.343,A -85,B 0,C 180,E1 -17549.825,E2 -17549.825} C_VEL
LIN {X 0,Y 288.327,Z 446.212,A -85,B 0,C 180,E1 -17550.294,E2 -17550.294} C_VEL
LIN {X 0,Y 288.922,Z 430.041,A -85,B 0,C 180,E1 -17550.767,E2 -17550.767} C_VEL
LIN {X 0,Y 290.505,Z 373.265,A -85,B 0,C 180,E1 -17552.196,E2 -17552.196} C_VEL
LIN {X 0,Y 287.795,Z 358.689,A -85,B 0,C 180,E1 -17552.837,E2 -17552.837} C_VEL
LIN {X 0,Y 281.147,Z 341.396,A -85,B 0,C 180,E1 -17553.945,E2 -17553.945} C_VEL
LIN {X 0,Y 279.21,Z 336.665,A -85,B 0,C 180,E1 -17554.331,E2 -17554.331} C_VEL
LIN {X 0,Y 277.664,Z 328.636,A -85,B 0,C 180,E1 -17557.362,E2 -17557.362} C_VEL
LIN {X 0,Y 277.562,Z 328.404,A -85,B 0,C 180,E1 -17559.069,E2 -17559.069} C_VEL
LIN {X 0,Y 277.418,Z 328.425,A -85,B 0,C 180,E1 -17563.18,E2 -17563.18} C_VEL
LIN {X 0,Y 277.407,Z 328.426,A -85,B 0,C 180,E1 -17566.182,E2 -17566.182} C_VEL
LIN {X 0,Y 277.346,Z 328.435,A -85,B 0,C 180,E1 -17570.349,E2 -17570.349} C_VEL
LIN {X 0,Y 277.294,Z 328.436,A -85,B 0,C 180,E1 -17574.158,E2 -17574.158} C_VEL
LIN {X 0,Y 277.326,Z 328.428,A -85,B 0,C 180,E1 -17577.505,E2 -17577.505} C_VEL
LIN {X 0,Y 277.274,Z 328.444,A -85,B 0,C 180,E1 -17580.481,E2 -17580.481} C_VEL
LIN {X 0,Y 277.256,Z 328.43,A -85,B 0,C 180,E1 -17583.895,E2 -17583.895} C_VEL
LIN {X 0,Y 277.283,Z 328.445,A -85,B 0,C 180,E1 -17587.467,E2 -17587.467} C_VEL
LIN {X 0,Y 277.212,Z 328.432,A -85,B 0,C 180,E1 -17591.236,E2 -17591.236} C_VEL
LIN {X 0,Y 277.219,Z 328.452,A -85,B 0,C 180,E1 -17595.223,E2 -17595.223} C_VEL
LIN {X 0,Y 277.223,Z 328.427,A -85,B 0,C 180,E1 -17599.512,E2 -17599.512} C_VEL
LIN {X 0,Y 277.262,Z 328.432,A -85,B 0,C 180,E1 -17602.53,E2 -17602.53} C_VEL
LIN {X 0,Y 277.249,Z 328.446,A -85,B 0,C 180,E1 -17606.104,E2 -17606.104} C_VEL
LIN {X 0,Y 277.264,Z 328.415,A -85,B 0,C 180,E1 -17609.539,E2 -17609.539} C_VEL
LIN {X 0,Y 277.256,Z 328.437,A -85,B 0,C 180,E1 -17613.908,E2 -17613.908} C_VEL
LIN {X 0,Y 277.268,Z 328.443,A -85,B 0,C 180,E1 -17617.653,E2 -17617.653} C_VEL
LIN {X 0,Y 277.304,Z 328.413,A -85,B 0,C 180,E1 -17620.202,E2 -17620.202} C_VEL
LIN {X 0,Y 276.657,Z 328.483,A -85,B 0,C 180,E1 -17621.415,E2 -17621.415} C_VEL
LIN {X 0,Y 273.853,Z 328.845,A -85,B 0,C 180,E1 -17623.394,E2 -17623.394} C_VEL
LIN {X 0,Y 271.465,Z 329.159,A -85,B 0,C 180,E1 -17625.001,E2 -17625.001} C_VEL
LIN {X 0,Y 270.434,Z 329.293,A -85,B 0,C 180,E1 -17626.245,E2 -17626.245} C_VEL
LIN {X 0,Y 270.347,Z 329.302,A -85,B 0,C 180,E1 -17626.667,E2 -17626.667} C_VEL
LIN {X 0,Y 270.529,Z 329.267,A -85,B 0,C 180,E1 -17631.032,E2 -17631.032} C_VEL
LIN {X 0,Y 270.512,Z 329.247,A -85,B 0,C 180,E1 -17634.035,E2 -17634.035} C_VEL
LIN {X 0,Y 270.772,Z 329.255,A -85,B 0,C 180,E1 -17638.512,E2 -17638.512} C_VEL
LIN {X 0,Y 270.777,Z 329.246,A -85,B 0,C 180,E1 -17641.487,E2 -17641.487} C_VEL
LIN {X 0,Y 270.576,Z 329.266,A -85,B 0,C 180,E1 -17647.462,E2 -17647.462} C_VEL
LIN {X 0,Y 270.407,Z 329.3,A -85,B 0,C 180,E1 -17650.482,E2 -17650.482} C_VEL
LIN {X 0,Y 270.339,Z 329.278,A -85,B 0,C 180,E1 -17655.068,E2 -17655.068} C_VEL
LIN {X 0,Y 270.222,Z 329.325,A -85,B 0,C 180,E1 -17659.761,E2 -17659.761} C_VEL
LIN {X 0,Y 270.224,Z 329.302,A -85,B 0,C 180,E1 -17664.59,E2 -17664.59} C_VEL
LIN {X 0,Y 270.198,Z 329.326,A -85,B 0,C 180,E1 -17667.916,E2 -17667.916} C_VEL
LIN {X 0,Y 270.173,Z 329.313,A -85,B 0,C 180,E1 -17671.349,E2 -17671.349} C_VEL
LIN {X 0,Y 270.197,Z 329.329,A -85,B 0,C 180,E1 -17674.906,E2 -17674.906} C_VEL
LIN {X 0,Y 270.167,Z 329.327,A -85,B 0,C 180,E1 -17678.702,E2 -17678.702} C_VEL
LIN {X 0,Y 270.146,Z 329.327,A -85,B 0,C 180,E1 -17683.244,E2 -17683.244} C_VEL
LIN {X 0,Y 270.149,Z 329.334,A -85,B 0,C 180,E1 -17687.437,E2 -17687.437} C_VEL
LIN {X 0,Y 270.206,Z 329.325,A -85,B 0,C 180,E1 -17691.374,E2 -17691.374} C_VEL
LIN {X 0,Y 270.221,Z 329.357,A -85,B 0,C 180,E1 -17695.734,E2 -17695.734} C_VEL
LIN {X 0,Y 271.386,Z 334.741,A -85,B 0,C 180,E1 -17697.915,E2 -17697.915} C_VEL
LIN {X 0,Y 273.203,Z 343.436,A -85,B 0,C 180,E1 -17701.093,E2 -17701.093} C_VEL
LIN {X 0,Y 274.567,Z 347.233,A -85,B 0,C 180,E1 -17701.434,E2 -17701.434} C_VEL
LIN {X 0,Y 279.56,Z 360.372,A -85,B 0,C 180,E1 -17702.293,E2 -17702.293} C_VEL
LIN {X 0,Y 283.704,Z 386.85,A -85,B 0,C 180,E1 -17703.425,E2 -17703.425} C_VEL
LIN {X 0,Y 281.79,Z 449.365,A -85,B 0,C 180,E1 -17705.061,E2 -17705.061} C_VEL
LIN {X 0,Y 281.233,Z 459.238,A -85,B 0,C 180,E1 -17705.452,E2 -17705.452} C_VEL
LIN {X 0,Y 280.349,Z 469.851,A -85,B 0,C 180,E1 -17706.058,E2 -17706.058} C_VEL
LIN {X 0,Y 279.22,Z 480.091,A -85,B 0,C 180,E1 -17706.841,E2 -17706.841} C_VEL
LIN {X 0,Y 277.858,Z 490.725,A -85,B 0,C 180,E1 -17707.899,E2 -17707.899} C_VEL
LIN {X 0,Y 276.362,Z 500.69,A -85,B 0,C 180,E1 -17709.144,E2 -17709.144} C_VEL
LIN {X 0,Y 275.039,Z 509.002,A -85,B 0,C 180,E1 -17710.404,E2 -17710.404} C_VEL
LIN {X 0,Y 273.613,Z 517.87,A -85,B 0,C 180,E1 -17712.047,E2 -17712.047} C_VEL
LIN {X 0,Y 272.433,Z 524.575,A -85,B 0,C 180,E1 -17713.515,E2 -17713.515} C_VEL
LIN {X 0,Y 271.172,Z 531.589,A -85,B 0,C 180,E1 -17715.363,E2 -17715.363} C_VEL
LIN {X 0,Y 270.101,Z 537.442,A -85,B 0,C 180,E1 -17717.222,E2 -17717.222} C_VEL
LIN {X 0,Y 269.238,Z 543.119,A -85,B 0,C 180,E1 -17719.471,E2 -17719.471} C_VEL
LIN {X 0,Y 268.614,Z 547.578,A -85,B 0,C 180,E1 -17721.726,E2 -17721.726} C_VEL
LIN {X 0,Y 268.247,Z 550.952,A -85,B 0,C 180,E1 -17723.984,E2 -17723.984} C_VEL
LIN {X 0,Y 268.141,Z 552.583,A -85,B 0,C 180,E1 -17725.49,E2 -17725.49} C_VEL
LIN {X 0,Y 268.124,Z 554.75,A -85,B 0,C 180,E1 -17728.498,E2 -17728.498} C_VEL
LIN {X 0,Y 268.125,Z 555.142,A -85,B 0,C 180,E1 -17731.502,E2 -17731.502} C_VEL
LIN {X 0,Y 268.112,Z 554.807,A -85,B 0,C 180,E1 -17733.005,E2 -17733.005} C_VEL
LIN {X 0,Y 268.301,Z 552.859,A -85,B 0,C 180,E1 -17736.014,E2 -17736.014} C_VEL
LIN {X 0,Y 268.687,Z 550.322,A -85,B 0,C 180,E1 -17738.271,E2 -17738.271} C_VEL
LIN {X 0,Y 269.344,Z 546.771,A -85,B 0,C 180,E1 -17740.524,E2 -17740.524} C_VEL
LIN {X 0,Y 270.336,Z 542.121,A -85,B 0,C 180,E1 -17742.766,E2 -17742.766} C_VEL
LIN {X 0,Y 271.739,Z 536.222,A -85,B 0,C 180,E1 -17744.989,E2 -17744.989} C_VEL
LIN {X 0,Y 273.507,Z 528.861,A -85,B 0,C 180,E1 -17747.188,E2 -17747.188} C_VEL
LIN {X 0,Y 275.052,Z 521.393,A -85,B 0,C 180,E1 -17749.021,E2 -17749.021} C_VEL
LIN {X 0,Y 276.824,Z 513.422,A -85,B 0,C 180,E1 -17750.625,E2 -17750.625} C_VEL
LIN {X 0,Y 278.59,Z 504.934,A -85,B 0,C 180,E1 -17752.04,E2 -17752.04} C_VEL
LIN {X 0,Y 280.345,Z 496.064,A -85,B 0,C 180,E1 -17753.256,E2 -17753.256} C_VEL
LIN {X 0,Y 282.205,Z 485.071,A -85,B 0,C 180,E1 -17754.458,E2 -17754.458} C_VEL
LIN {X 0,Y 283.535,Z 475.283,A -85,B 0,C 180,E1 -17755.314,E2 -17755.314} C_VEL
LIN {X 0,Y 284.84,Z 463.662,A -85,B 0,C 180,E1 -17756.072,E2 -17756.072} C_VEL
LIN {X 0,Y 285.819,Z 453.29,A -85,B 0,C 180,E1 -17756.542,E2 -17756.542} C_VEL
LIN {X 0,Y 286.446,Z 436.08,A -85,B 0,C 180,E1 -17757.064,E2 -17757.064} C_VEL
LIN {X 0,Y 288.085,Z 387.404,A -85,B 0,C 180,E1 -17758.325,E2 -17758.325} C_VEL
LIN {X 0,Y 284.792,Z 367.395,A -85,B 0,C 180,E1 -17759.35,E2 -17759.35} C_VEL
LIN {X 0,Y 278.519,Z 353.068,A -85,B 0,C 180,E1 -17760.65,E2 -17760.65} C_VEL
LIN {X 0,Y 273.688,Z 342.94,A -85,B 0,C 180,E1 -17761.718,E2 -17761.718} C_VEL
LIN {X 0,Y 272.952,Z 340.026,A -85,B 0,C 180,E1 -17762.732,E2 -17762.732} C_VEL
LIN {X 0,Y 270.719,Z 331.161,A -85,B 0,C 180,E1 -17766.412,E2 -17766.412} C_VEL
LIN {X 0,Y 270.233,Z 329.344,A -85,B 0,C 180,E1 -17767.351,E2 -17767.351} C_VEL
LIN {X 0,Y 270.167,Z 329.32,A -85,B 0,C 180,E1 -17771.028,E2 -17771.028} C_VEL
LIN {X 0,Y 270.15,Z 329.331,A -85,B 0,C 180,E1 -17775.38,E2 -17775.38} C_VEL
LIN {X 0,Y 270.172,Z 329.329,A -85,B 0,C 180,E1 -17779.434,E2 -17779.434} C_VEL
LIN {X 0,Y 270.224,Z 329.323,A -85,B 0,C 180,E1 -17783.731,E2 -17783.731} C_VEL
LIN {X 0,Y 270.202,Z 329.327,A -85,B 0,C 180,E1 -17786.893,E2 -17786.893} C_VEL
LIN {X 0,Y 270.219,Z 329.326,A -85,B 0,C 180,E1 -17790.386,E2 -17790.386} C_VEL
LIN {X 0,Y 270.263,Z 329.316,A -85,B 0,C 180,E1 -17793.764,E2 -17793.764} C_VEL
LIN {X 0,Y 270.233,Z 329.313,A -85,B 0,C 180,E1 -17797.039,E2 -17797.039} C_VEL
LIN {X 0,Y 270.302,Z 329.312,A -85,B 0,C 180,E1 -17800.245,E2 -17800.245} C_VEL
LIN {X 0,Y 270.403,Z 329.298,A -85,B 0,C 180,E1 -17804.936,E2 -17804.936} C_VEL
LIN {X 0,Y 270.442,Z 329.294,A -85,B 0,C 180,E1 -17809.519,E2 -17809.519} C_VEL
LIN {X 0,Y 270.613,Z 329.273,A -85,B 0,C 180,E1 -17812.539,E2 -17812.539} C_VEL
LIN {X 0,Y 270.789,Z 329.254,A -85,B 0,C 180,E1 -17818.513,E2 -17818.513} C_VEL
LIN {X 0,Y 270.789,Z 329.249,A -85,B 0,C 180,E1 -17821.488,E2 -17821.488} C_VEL
LIN {X 0,Y 270.613,Z 329.274,A -85,B 0,C 180,E1 -17827.461,E2 -17827.461} C_VEL
LIN {X 0,Y 270.443,Z 329.297,A -85,B 0,C 180,E1 -17830.481,E2 -17830.481} C_VEL
LIN {X 0,Y 270.404,Z 329.301,A -85,B 0,C 180,E1 -17835.065,E2 -17835.065} C_VEL
LIN {X 0,Y 270.301,Z 329.311,A -85,B 0,C 180,E1 -17839.756,E2 -17839.756} C_VEL
LIN {X 0,Y 270.234,Z 329.321,A -85,B 0,C 180,E1 -17844.59,E2 -17844.59} C_VEL
LIN {X 0,Y 270.244,Z 329.307,A -85,B 0,C 180,E1 -17847.912,E2 -17847.912} C_VEL
LIN {X 0,Y 270.247,Z 329.461,A -85,B 0,C 180,E1 -17851.112,E2 -17851.112} C_VEL
LIN {X 0,Y 272.176,Z 336.419,A -85,B 0,C 180,E1 -17854.027,E2 -17854.027} C_VEL
LIN {X 0,Y 274.15,Z 340.387,A -85,B 0,C 180,E1 -17854.555,E2 -17854.555} C_VEL
LIN {X 0,Y 281.407,Z 354.931,A -85,B 0,C 180,E1 -17856.055,E2 -17856.055} C_VEL
LIN {X 0,Y 287.357,Z 369.148,A -85,B 0,C 180,E1 -17857.28,E2 -17857.28} C_VEL
LIN {X 0,Y 288.539,Z 375.918,A -85,B 0,C 180,E1 -17857.631,E2 -17857.631} C_VEL
LIN {X 0,Y 286.069,Z 442.083,A -85,B 0,C 180,E1 -17859.354,E2 -17859.354} C_VEL
LIN {X 0,Y 285.349,Z 452.647,A -85,B 0,C 180,E1 -17859.771,E2 -17859.771} C_VEL
LIN {X 0,Y 284.348,Z 463.418,A -85,B 0,C 180,E1 -17860.398,E2 -17860.398} C_VEL
LIN {X 0,Y 283.129,Z 473.689,A -85,B 0,C 180,E1 -17861.198,E2 -17861.198} C_VEL
LIN {X 0,Y 281.711,Z 483.195,A -85,B 0,C 180,E1 -17862.131,E2 -17862.131} C_VEL
LIN {X 0,Y 280.087,Z 492.797,A -85,B 0,C 180,E1 -17863.308,E2 -17863.308} C_VEL
LIN {X 0,Y 278.257,Z 502.237,A -85,B 0,C 180,E1 -17864.736,E2 -17864.736} C_VEL
LIN {X 0,Y 276.544,Z 510.121,A -85,B 0,C 180,E1 -17866.17,E2 -17866.17} C_VEL
LIN {X 0,Y 274.751,Z 517.9,A -85,B 0,C 180,E1 -17867.886,E2 -17867.886} C_VEL
LIN {X 0,Y 273.002,Z 525.439,A -85,B 0,C 180,E1 -17869.941,E2 -17869.941} C_VEL
LIN {X 0,Y 271.735,Z 530.624,A -85,B 0,C 180,E1 -17871.631,E2 -17871.631} C_VEL
LIN {X 0,Y 270.557,Z 535.65,A -85,B 0,C 180,E1 -17873.635,E2 -17873.635} C_VEL
LIN {X 0,Y 269.5,Z 540.11,A -85,B 0,C 180,E1 -17875.899,E2 -17875.899} C_VEL
LIN {X 0,Y 268.683,Z 543.791,A -85,B 0,C 180,E1 -17878.457,E2 -17878.457} C_VEL
LIN {X 0,Y 268.31,Z 545.603,A -85,B 0,C 180,E1 -17880.154,E2 -17880.154} C_VEL
LIN {X 0,Y 267.856,Z 547.39,A -85,B 0,C 180,E1 -17883.138,E2 -17883.138} C_VEL
LIN {X 0,Y 267.742,Z 547.777,A -85,B 0,C 180,E1 -17885.166,E2 -17885.166} C_VEL
LIN {X 0,Y 267.737,Z 547.435,A -85,B 0,C 180,E1 -17886.812,E2 -17886.812} C_VEL
LIN {X 0,Y 267.962,Z 545.593,A -85,B 0,C 180,E1 -17890.065,E2 -17890.065} C_VEL
LIN {X 0,Y 268.423,Z 542.899,A -85,B 0,C 180,E1 -17892.476,E2 -17892.476} C_VEL
LIN {X 0,Y 269.05,Z 538.538,A -85,B 0,C 180,E1 -17895.128,E2 -17895.128} C_VEL
LIN {X 0,Y 269.904,Z 533.08,A -85,B 0,C 180,E1 -17897.595,E2 -17897.595} C_VEL
LIN {X 0,Y 270.81,Z 527.707,A -85,B 0,C 180,E1 -17899.534,E2 -17899.534} C_VEL
LIN {X 0,Y 272.016,Z 521.188,A -85,B 0,C 180,E1 -17901.457,E2 -17901.457} C_VEL
LIN {X 0,Y 273.155,Z 515.064,A -85,B 0,C 180,E1 -17902.98,E2 -17902.98} C_VEL
LIN {X 0,Y 274.63,Z 506.29,A -85,B 0,C 180,E1 -17904.778,E2 -17904.778} C_VEL
LIN {X 0,Y 276.023,Z 498.093,A -85,B 0,C 180,E1 -17906.168,E2 -17906.168} C_VEL
LIN {X 0,Y 277.426,Z 488.876,A -85,B 0,C 180,E1 -17907.459,E2 -17907.459} C_VEL
LIN {X 0,Y 278.716,Z 479.297,A -85,B 0,C 180,E1 -17908.555,E2 -17908.555} C_VEL
LIN {X 0,Y 280.014,Z 468.16,A -85,B 0,C 180,E1 -17909.551,E2 -17909.551} C_VEL
LIN {X 0,Y 280.973,Z 456.525,A -85,B 0,C 180,E1 -17910.336,E2 -17910.336} C_VEL
LIN {X 0,Y 281.764,Z 446.054,A -85,B 0,C 180,E1 -17910.827,E2 -17910.827} C_VEL
LIN {X 0,Y 282.362,Z 430.003,A -85,B 0,C 180,E1 -17911.306,E2 -17911.306} C_VEL
LIN {X 0,Y 284.027,Z 374.335,A -85,B 0,C 180,E1 -17912.734,E2 -17912.734} C_VEL
LIN {X 0,Y 281.445,Z 360.662,A -85,B 0,C 180,E1 -17913.361,E2 -17913.361} C_VEL
LIN {X 0,Y 274.745,Z 343.349,A -85,B 0,C 180,E1 -17914.511,E2 -17914.511} C_VEL
LIN {X 0,Y 272.037,Z 336.884,A -85,B 0,C 180,E1 -17915.03,E2 -17915.03} C_VEL
LIN {X 0,Y 270.825,Z 330.482,A -85,B 0,C 180,E1 -17917.455,E2 -17917.455} C_VEL
LIN {X 0,Y 270.549,Z 329.298,A -85,B 0,C 180,E1 -17918.106,E2 -17918.106} C_VEL
LIN {X 0,Y 270.379,Z 329.294,A -85,B 0,C 180,E1 -17922.002,E2 -17922.002} C_VEL
LIN {X 0,Y 270.383,Z 329.299,A -85,B 0,C 180,E1 -17925.901,E2 -17925.901} C_VEL
LIN {X 0,Y 270.293,Z 329.317,A -85,B 0,C 180,E1 -17930.601,E2 -17930.601} C_VEL
LIN {X 0,Y 270.24,Z 329.318,A -85,B 0,C 180,E1 -17934.589,E2 -17934.589} C_VEL
LIN {X 0,Y 270.272,Z 329.305,A -85,B 0,C 180,E1 -17937.909,E2 -17937.909} C_VEL
LIN {X 0,Y 270.186,Z 329.331,A -85,B 0,C 180,E1 -17941.348,E2 -17941.348} C_VEL
LIN {X 0,Y 270.217,Z 329.307,A -85,B 0,C 180,E1 -17944.904,E2 -17944.904} C_VEL
LIN {X 0,Y 270.224,Z 329.322,A -85,B 0,C 180,E1 -17948.717,E2 -17948.717} C_VEL
LIN {X 0,Y 270.173,Z 329.318,A -85,B 0,C 180,E1 -17953.25,E2 -17953.25} C_VEL
LIN {X 0,Y 270.176,Z 329.324,A -85,B 0,C 180,E1 -17957.442,E2 -17957.442} C_VEL
LIN {X 0,Y 270.209,Z 329.299,A -85,B 0,C 180,E1 -17961.374,E2 -17961.374} C_VEL
LIN {X 0,Y 270.203,Z 329.326,A -85,B 0,C 180,E1 -17965.094,E2 -17965.094} C_VEL
LIN {X 0,Y 270.186,Z 329.301,A -85,B 0,C 180,E1 -17969.136,E2 -17969.136} C_VEL
LIN {X 0,Y 270.225,Z 329.295,A -85,B 0,C 180,E1 -17972.162,E2 -17972.162} C_VEL
LIN {X 0,Y 270.233,Z 329.32,A -85,B 0,C 180,E1 -17975.541,E2 -17975.541} C_VEL
LIN {X 0,Y 270.26,Z 329.288,A -85,B 0,C 180,E1 -17980.241,E2 -17980.241} C_VEL
LIN {X 0,Y 270.375,Z 329.289,A -85,B 0,C 180,E1 -17984.933,E2 -17984.933} C_VEL
LIN {X 0,Y 270.347,Z 329.302,A -85,B 0,C 180,E1 -17986.667,E2 -17986.667} C_VEL
LIN {X 0,Y 269.691,Z 329.39,A -85,B 0,C 180,E1 -17987.912,E2 -17987.912} C_VEL
LIN {X 0,Y 266.919,Z 329.725,A -85,B 0,C 180,E1 -17989.944,E2 -17989.944} C_VEL
LIN {X 0,Y 264.57,Z 330.001,A -85,B 0,C 180,E1 -17991.595,E2 -17991.595} C_VEL
LIN {X 0,Y 263.562,Z 330.114,A -85,B 0,C 180,E1 -17992.873,E2 -17992.873} C_VEL
LIN {X 0,Y 263.478,Z 330.122,A -85,B 0,C 180,E1 -17993.306,E2 -17993.306} C_VEL
